(* Logix 5000 project; controller Hose_HP_Test_Rig_V1 vendor 1 type 14 code 149 rev 32.11; software revision 32.00; part 2 of 10 *)

ADD_ON_INSTRUCTION SA_SOL_FWD_RET_SEQ   (* revision 1.0 *)
VAR_INPUT
   SA_SOL_SEQ : DINT; {required}
END_VAR
VAR_OUTPUT
   SA_SOL_SOL : BOOL; {required}
END_VAR
VAR_INPUT
   SA_SOL_PS : BOOL; {required}
END_VAR
VAR_OUTPUT
   SA_FWD_PS_OK : BOOL; {access None, required}
   SA_SOL_PS_FLT : BOOL; {required}
END_VAR
VAR_INPUT
   FLT_RST_PB : BOOL; {required}
   MSG_CODE : DINT; {required}
   FLT_CODE : DINT; {required}
END_VAR
VAR_OUTPUT
   ERROR_CODE : DINT; {required}
END_VAR
VAR_INPUT
   SEQ_NO : DINT;
   SA_RET_PS : BOOL; {required}
END_VAR
VAR_OUTPUT
   SA_RET_PS_OK : BOOL; {required}
END_VAR
VAR
   SA_SOL_SEQ_ON : BOOL; {access None}
   DA_SOL_PS_FAULT : TIMER; {access None}
   SA_SOL_PS_FAULT : TIMER := (PRE := 3000); {access None}
END_VAR

ROUTINE Logic   (* ladder *)
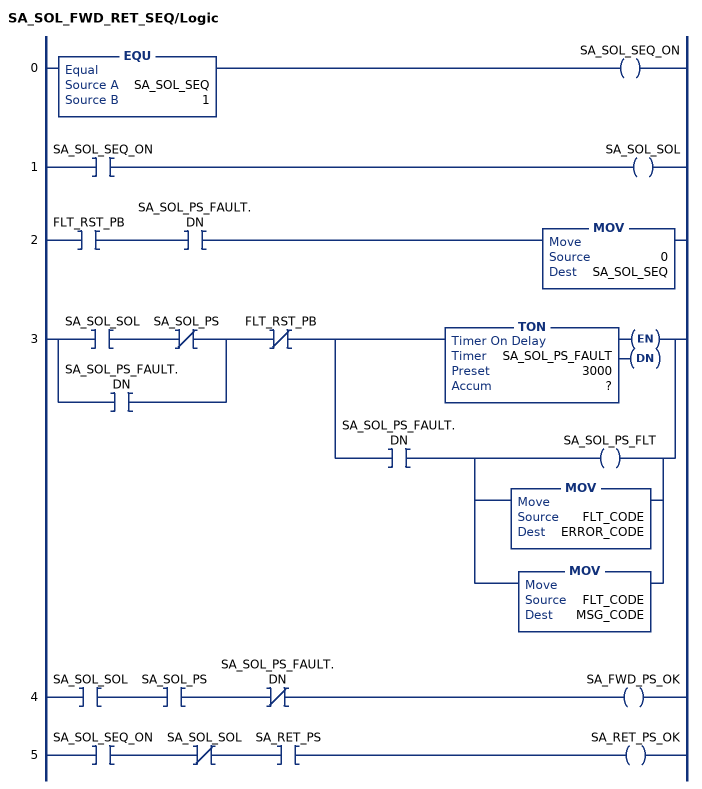
   0: EQU(SA_SOL_SEQ,1)OTE(SA_SOL_SEQ_ON);
   1: XIC(SA_SOL_SEQ_ON)OTE(SA_SOL_SOL);
   2: XIC(FLT_RST_PB)XIC(SA_SOL_PS_FAULT.DN)MOV(0,SA_SOL_SEQ);
   3: [XIC(SA_SOL_SOL) XIO(SA_SOL_PS) ,XIC(SA_SOL_PS_FAULT.DN) ]XIO(FLT_RST_PB)[TON(SA_SOL_PS_FAULT,?,?) ,XIC(SA_SOL_PS_FAULT.DN) [OTE(SA_SOL_PS_FLT) ,MOV(FLT_CODE,ERROR_CODE) ,MOV(FLT_CODE,MSG_CODE) ] ];
   4: XIC(SA_SOL_SOL)XIC(SA_SOL_PS)XIO(SA_SOL_PS_FAULT.DN)OTE(SA_FWD_PS_OK);
   5: XIC(SA_SOL_SEQ_ON)XIO(SA_SOL_SOL)XIC(SA_RET_PS)OTE(SA_RET_PS_OK);
END_ROUTINE
END_ADD_ON_INSTRUCTION

ADD_ON_INSTRUCTION SCP   (* revision 1.0 *)
VAR_OUTPUT
   Y : REAL; {access Read Only, required}
END_VAR
VAR_INPUT
   X : REAL; {required}
   X1 : REAL; {required}
   X2 : REAL; {required}
   Y1 : REAL; {required}
   Y2 : REAL; {required}
   C : REAL; {required}
END_VAR

ROUTINE Logic   (* structured text *)
   Y:=((X-X1)*((Y2-Y1)/(X2-X1))+Y1)+C;
END_ROUTINE
END_ADD_ON_INSTRUCTION

ADD_ON_INSTRUCTION SEQ_START_AND_FILL   (* revision 1.0 *)
VAR_INPUT
   SET_SEQ_NO : DINT; {required}
END_VAR
VAR_IN_OUT
   CURR_SEQ_NO : DINT; {required}
END_VAR
VAR_OUTPUT
   EXHS_VAL_ON : BOOL; {required}
   TEST_VAL_ON : BOOL; {required}
END_VAR
VAR_INPUT
   TEST_VAL_OFF : BOOL; {required}
   FAULTED : BOOL; {required}
   RST_TEST_VAL_OFF : BOOL; {required}
   EXHS_VAL_OFF : BOOL; {required}
   RST_EXHS_VAL_OFF : BOOL; {required}
END_VAR
VAR_IN_OUT
   TEST_STS : DINT; {required}
END_VAR
VAR_INPUT
   NEXT_SEQ_NO : DINT; {required}
END_VAR
VAR
   SEQ_START : BOOL; {access None}
   ONS1 : BOOL; {access None}
   ONS2 : BOOL; {access None}
   TEST_VAL_ON_DEL : TIMER := (PRE := 500); {access None}
   ONS3 : BOOL; {access None}
   EXHS_VAL_DEL : TIMER := (PRE := 250); {access None}
END_VAR

ROUTINE Logic   (* ladder *)
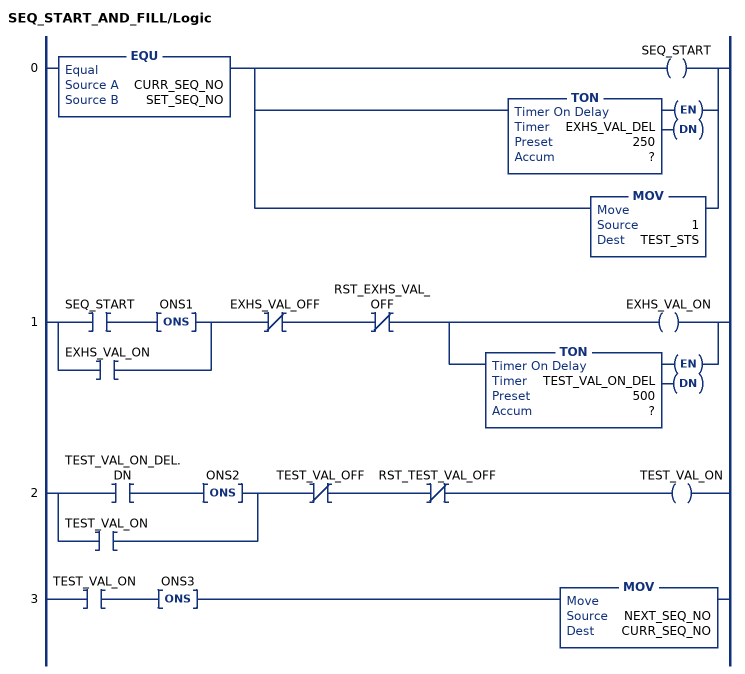
   0: EQU(CURR_SEQ_NO,SET_SEQ_NO)[OTE(SEQ_START) ,TON(EXHS_VAL_DEL,?,?) ,MOV(1,TEST_STS) ];
   1: [XIC(SEQ_START) ONS(ONS1) ,XIC(EXHS_VAL_ON) ]XIO(EXHS_VAL_OFF)XIO(RST_EXHS_VAL_OFF)[OTE(EXHS_VAL_ON) ,TON(TEST_VAL_ON_DEL,?,?) ];
   2: [XIC(TEST_VAL_ON_DEL.DN) ONS(ONS2) ,XIC(TEST_VAL_ON) ]XIO(TEST_VAL_OFF)XIO(RST_TEST_VAL_OFF)OTE(TEST_VAL_ON);
   3: XIC(TEST_VAL_ON)ONS(ONS3)MOV(NEXT_SEQ_NO,CURR_SEQ_NO);
END_ROUTINE
END_ADD_ON_INSTRUCTION

ADD_ON_INSTRUCTION SETTING_MODE   (* revision 1.0 *)
VAR_IN_OUT
   CURRENT_SCREEN : DINT; {required}
END_VAR
VAR_INPUT
   SET_MODE_SCREEN : DINT; {required}
   CALB_MODE_SCREEN : BOOL; {required}
END_VAR
VAR_OUTPUT
   SET_MODE_SEL : BOOL; {required}
END_VAR
VAR_INPUT
   LH_START_PB : BOOL; {required}
   TOP_CLAMP_SEL : BOOL; {required}
END_VAR
VAR_OUTPUT
   TOP_CLAMP_SET : BOOL; {required}
   TOP_DECLAMP_SET : BOOL; {required}
END_VAR
VAR_INPUT
   RST_SEQ_ON : BOOL; {required}
   BOTTOM_CLAMP_SEL : BOOL; {required}
END_VAR
VAR_OUTPUT
   BOTTOM_DECLAMP_SET : BOOL; {required}
   BOTTOM_CLAMP_SET : BOOL; {required}
END_VAR
VAR_INPUT
   DOOR_CLOSE_SEL : BOOL; {required}
END_VAR
VAR_OUTPUT
   DOOR_CLOSE_SET : BOOL; {required}
   DOOR_OPEN_SET : BOOL; {required}
END_VAR
VAR
   ONS1 : BOOL; {access None}
   SET_PB_ONS : BOOL; {access None}
   TOP_DECLAMP_OFF_DEL : TIMER := (PRE := 250); {access None}
   BOTTOM_DECLAMP_OFF_DEL : TIMER := (PRE := 250); {access None}
   DOOR_OPEN_OFF_DEL : TIMER := (PRE := 250); {access None}
   ons2 : BOOL; {access None}
END_VAR

ROUTINE Logic   (* ladder *)
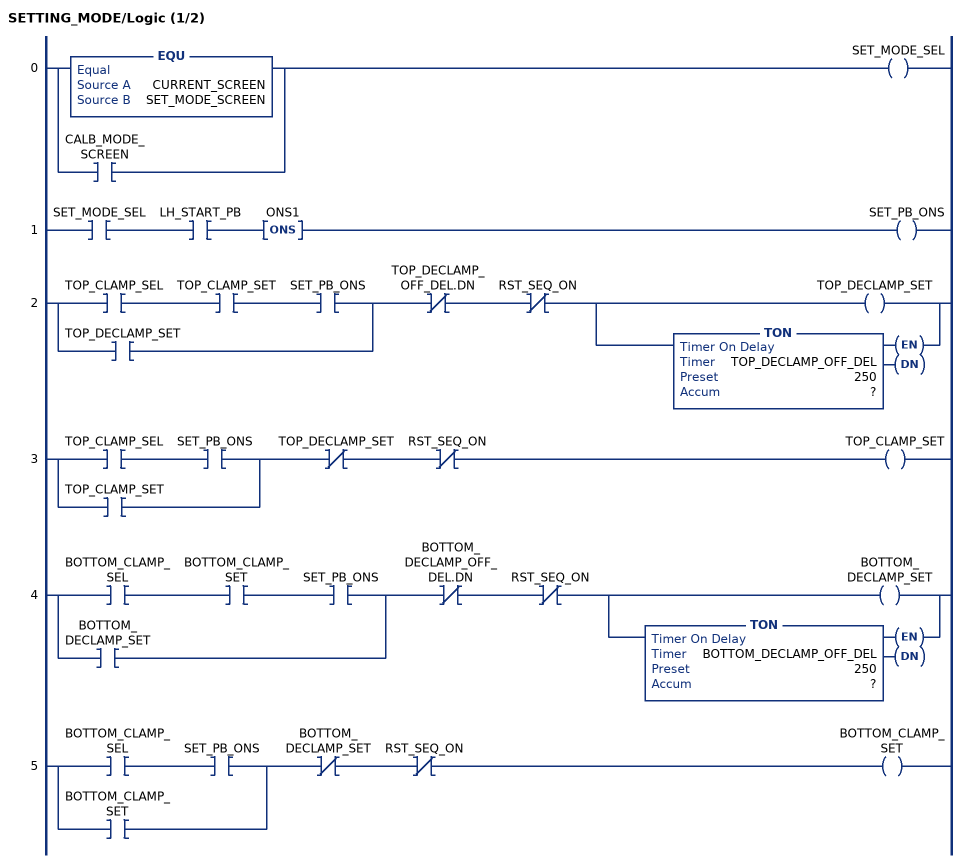
   0: [EQU(CURRENT_SCREEN,SET_MODE_SCREEN) ,XIC(CALB_MODE_SCREEN) ]OTE(SET_MODE_SEL);
   1: XIC(SET_MODE_SEL)XIC(LH_START_PB)ONS(ONS1)OTE(SET_PB_ONS);
   2: [XIC(TOP_CLAMP_SEL) XIC(TOP_CLAMP_SET) XIC(SET_PB_ONS) ,XIC(TOP_DECLAMP_SET) ]XIO(TOP_DECLAMP_OFF_DEL.DN)XIO(RST_SEQ_ON)[OTE(TOP_DECLAMP_SET) ,TON(TOP_DECLAMP_OFF_DEL,?,?) ];
   3: [XIC(TOP_CLAMP_SEL) XIC(SET_PB_ONS) ,XIC(TOP_CLAMP_SET) ]XIO(TOP_DECLAMP_SET)XIO(RST_SEQ_ON)OTE(TOP_CLAMP_SET);
   4: [XIC(BOTTOM_CLAMP_SEL) XIC(BOTTOM_CLAMP_SET) XIC(SET_PB_ONS) ,XIC(BOTTOM_DECLAMP_SET) ]XIO(BOTTOM_DECLAMP_OFF_DEL.DN)XIO(RST_SEQ_ON)[OTE(BOTTOM_DECLAMP_SET) ,TON(BOTTOM_DECLAMP_OFF_DEL,?,?) ];
   5: [XIC(BOTTOM_CLAMP_SEL) XIC(SET_PB_ONS) ,XIC(BOTTOM_CLAMP_SET) ]XIO(BOTTOM_DECLAMP_SET)XIO(RST_SEQ_ON)OTE(BOTTOM_CLAMP_SET);
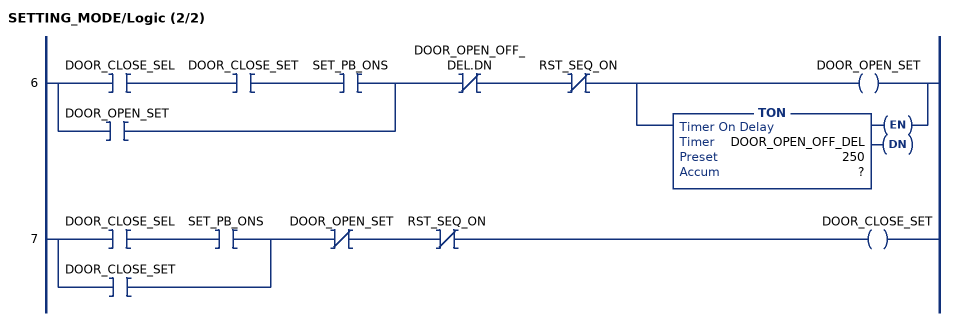
   6: [XIC(DOOR_CLOSE_SEL) XIC(DOOR_CLOSE_SET) XIC(SET_PB_ONS) ,XIC(DOOR_OPEN_SET) ]XIO(DOOR_OPEN_OFF_DEL.DN)XIO(RST_SEQ_ON)[OTE(DOOR_OPEN_SET) ,TON(DOOR_OPEN_OFF_DEL,?,?) ];
   7: [XIC(DOOR_CLOSE_SEL) XIC(SET_PB_ONS) ,XIC(DOOR_CLOSE_SET) ]XIO(DOOR_OPEN_SET)XIO(RST_SEQ_ON)OTE(DOOR_CLOSE_SET);
END_ROUTINE
END_ADD_ON_INSTRUCTION

ADD_ON_INSTRUCTION STAMP_SEQ   (* revision 1.0 *)
VAR_INPUT
   SET_SEQ_NO : DINT; {required}
END_VAR
VAR_IN_OUT
   CUR_SEQ_NO : DINT; {required}
END_VAR
VAR_OUTPUT
   STAMP_FWD_SOL : BOOL; {required}
END_VAR
VAR_INPUT
   STAMP_FWD_PS : BOOL; {required}
END_VAR
VAR_OUTPUT
   STAMP_FWD_OK : BOOL; {required}
   STAMP_NOT_FWD : BOOL; {required}
   STAMP_RET_OK : BOOL;
END_VAR
VAR_INPUT
   FLT_RST_PB : BOOL; {required}
   FAULTED : BOOL; {required}
   FLT_CODE : DINT; {required}
END_VAR
VAR_IN_OUT
   ERROR_CODE : DINT; {required}
END_VAR
VAR_INPUT
   RUN_CODE : DINT; {required}
END_VAR
VAR_IN_OUT
   MSG : DINT; {required}
END_VAR
VAR_INPUT
   NEXT_SEQ_NO : DINT; {required}
END_VAR
VAR
   STAMP_SEQ : BOOL; {access None}
   STAMP_PS_CHK_DEL : TIMER := (PRE := 3000); {access None}
   STAMP_PS_FWD_CHK : TIMER := (PRE := 500); {access None}
END_VAR

ROUTINE Logic   (* ladder *)
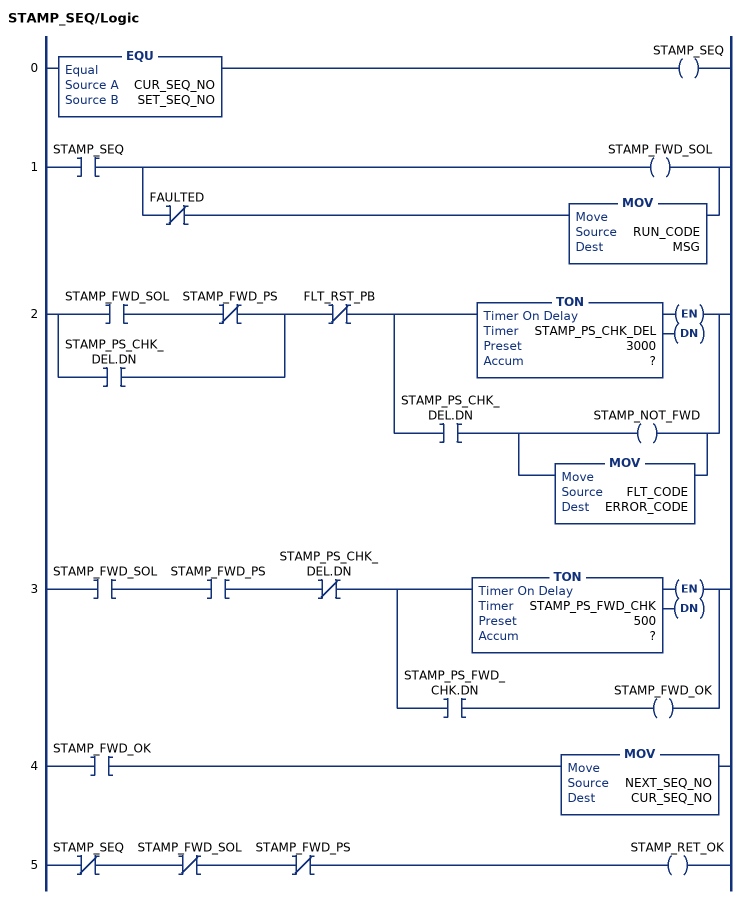
   0: EQU(CUR_SEQ_NO,SET_SEQ_NO)OTE(STAMP_SEQ);
   1: XIC(STAMP_SEQ)[OTE(STAMP_FWD_SOL) ,XIO(FAULTED) MOV(RUN_CODE,MSG) ];
   2: [XIC(STAMP_FWD_SOL) XIO(STAMP_FWD_PS) ,XIC(STAMP_PS_CHK_DEL.DN) ]XIO(FLT_RST_PB)[TON(STAMP_PS_CHK_DEL,?,?) ,XIC(STAMP_PS_CHK_DEL.DN) [OTE(STAMP_NOT_FWD) ,MOV(FLT_CODE,ERROR_CODE) ] ];
   3: XIC(STAMP_FWD_SOL)XIC(STAMP_FWD_PS)XIO(STAMP_PS_CHK_DEL.DN)[TON(STAMP_PS_FWD_CHK,?,?) ,XIC(STAMP_PS_FWD_CHK.DN) OTE(STAMP_FWD_OK) ];
   4: XIC(STAMP_FWD_OK)MOV(NEXT_SEQ_NO,CUR_SEQ_NO);
   5: XIO(STAMP_SEQ)XIO(STAMP_FWD_SOL)XIO(STAMP_FWD_PS)OTE(STAMP_RET_OK);
END_ROUTINE
END_ADD_ON_INSTRUCTION

ADD_ON_INSTRUCTION TEST_TAIL_END   (* revision 1.0 *)
VAR_INPUT
   SET_SEQ_NO : DINT; {required}
END_VAR
VAR_IN_OUT
   CUR_SEQ_NO : DINT; {required}
END_VAR
VAR_INPUT
   STN_ON : BOOL; {required}
   AUTO_MODE : BOOL; {required}
   POKAYOKE_NOT_DONE : BOOL; {required}
   PYOKE_LT : BOOL; {required}
   STAB_HIGH : BOOL; {required}
   STAB_LOW : BOOL; {required}
END_VAR
VAR_OUTPUT
   LT_COMPLETED : BOOL; {required}
END_VAR
VAR_INPUT
   LT_DROP_OK : BOOL; {required}
   DROP_NOK : BOOL; {required}
END_VAR
VAR_IN_OUT
   LT_POKEYOKE : DINT; {required}
   TEST_STS : DINT; {required}
END_VAR
VAR_INPUT
   NEXT_SEQ_NO : DINT; {required}
END_VAR

ROUTINE Logic   (* ladder *)
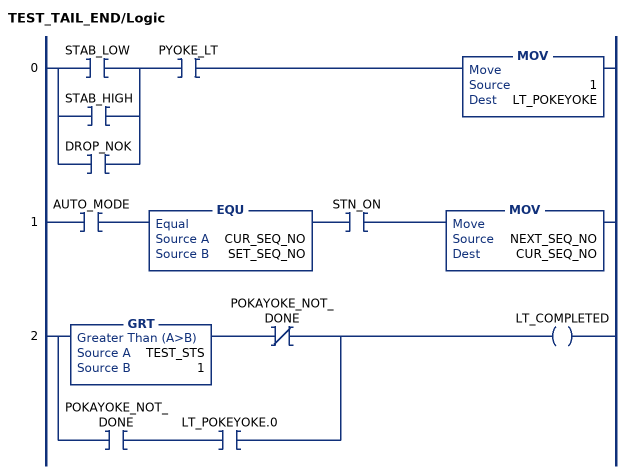
   0: [XIC(STAB_LOW) ,XIC(STAB_HIGH) ,XIC(DROP_NOK) ]XIC(PYOKE_LT)MOV(1,LT_POKEYOKE);
   1: XIC(AUTO_MODE)EQU(CUR_SEQ_NO,SET_SEQ_NO)XIC(STN_ON)MOV(NEXT_SEQ_NO,CUR_SEQ_NO);
   2: [GRT(TEST_STS,1) XIO(POKAYOKE_NOT_DONE) ,XIC(POKAYOKE_NOT_DONE) XIC(LT_POKEYOKE.0) ]OTE(LT_COMPLETED);
END_ROUTINE
END_ADD_ON_INSTRUCTION

ADD_ON_INSTRUCTION TOP_DECLAMP   (* revision 1.0 *)
VAR_INPUT
   SET_SEQ_NO : DINT; {required}
END_VAR
VAR_IN_OUT
   CUR_SEQ_NO : DINT; {required}
END_VAR
VAR_INPUT
   TEST_ON : BOOL; {required}
   FAULTED : BOOL; {required}
END_VAR
VAR_OUTPUT
   TOP_DECLAMP_AUTO : BOOL; {required}
   TOP_DECLAMP_OK : BOOL; {required}
END_VAR
VAR_INPUT
   TOP_CLAMP_PS : BOOL; {required}
   TOP_NOT_DECLAMPED : BOOL; {required}
   CONSTRICTION : BOOL; {required}
   NEXT_SEQ_NO : DINT; {required}
   END_SEQ_NO : DINT; {required}
END_VAR
VAR
   TOP_DECLAMP_SEQ_AUTO : BOOL; {access None}
   ONS1 : BOOL; {access None}
   TOP_DECLAMP_CHK_DEL : TIMER := (PRE := 500); {access None}
END_VAR

ROUTINE Logic   (* ladder *)
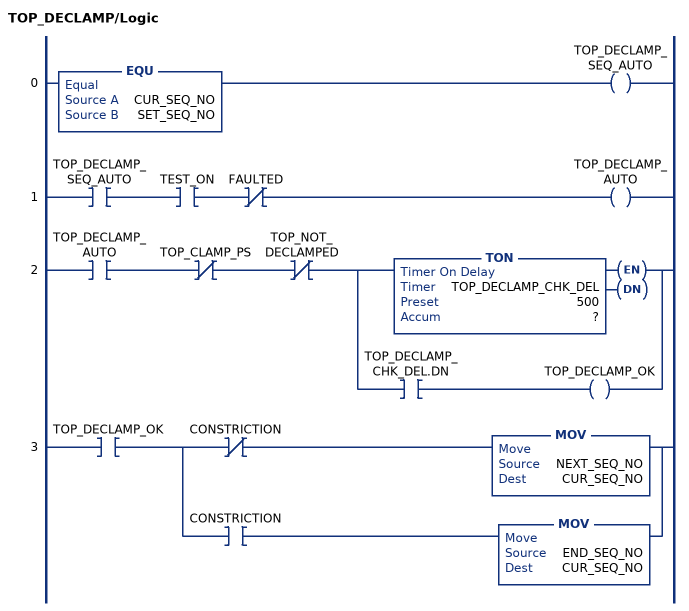
   0: EQU(CUR_SEQ_NO,SET_SEQ_NO)OTE(TOP_DECLAMP_SEQ_AUTO);
   1: XIC(TOP_DECLAMP_SEQ_AUTO)XIC(TEST_ON)XIO(FAULTED)OTE(TOP_DECLAMP_AUTO);
   2: XIC(TOP_DECLAMP_AUTO)XIO(TOP_CLAMP_PS)XIO(TOP_NOT_DECLAMPED)[TON(TOP_DECLAMP_CHK_DEL,?,?) ,XIC(TOP_DECLAMP_CHK_DEL.DN) OTE(TOP_DECLAMP_OK) ];
   3: XIC(TOP_DECLAMP_OK)[XIO(CONSTRICTION) MOV(NEXT_SEQ_NO,CUR_SEQ_NO) ,XIC(CONSTRICTION) MOV(END_SEQ_NO,CUR_SEQ_NO) ];
END_ROUTINE
END_ADD_ON_INSTRUCTION

ADD_ON_INSTRUCTION TS_TIMEOUT   (* revision 1.0 *)
VAR_IN_OUT
   TS_STS : DINT; {required}
END_VAR
VAR_INPUT
   CHECK_TRACE_STS : BOOL; {required}
   RETEST : BOOL; {required}
END_VAR
VAR_IN_OUT
   MSG : DINT; {required}
END_VAR
VAR_OUTPUT
   TS_TIMEOUT_FLT : BOOL; {access Read Only, required}
END_VAR
VAR
   TS_TIMEOUT : TIMER := (PRE := 3000); {access None}
END_VAR

ROUTINE Logic   (* ladder *)
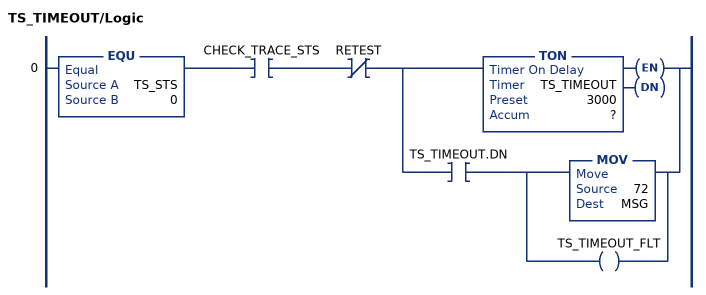
   0: EQU(TS_STS,0)XIC(CHECK_TRACE_STS)XIO(RETEST)[TON(TS_TIMEOUT,?,?) ,XIC(TS_TIMEOUT.DN) [MOV(72,MSG) ,OTE(TS_TIMEOUT_FLT) ] ];
END_ROUTINE
END_ADD_ON_INSTRUCTION

VAR_GLOBAL   (* controller tags *)
   ABORT_STN1 : BOOL;
   ABORT_STN2 : BOOL;
   ABORT_STN3 : BOOL;
   ABORT_STN4 : BOOL;
   ACT_DROP_STN1 : REAL := 0.49569702;
   ACT_DROP_STN2 : REAL := 0.5277252;
   ACT_DROP_STN3 : REAL := 0.5121765;
   ACT_DROP_STN4 : REAL := 0.4958496;
   ACT_PR_STN1 : REAL := -0.05;
   ACT_PR_STN2 : REAL := -0.015992021;
   ACT_PR_STN3 : REAL;
   ACT_PR_STN4 : REAL := 0.015994694;
   ACT_TRAVEL : REAL := 9187.228;
   AUTO_DOOR_OPEN_BLK_STN1 : DA_SOL_RET_SEQ := (FWD_SOL_PS := 1, RUN_CODE := 3, FLT_CODE := 18, SET_SEQ_NO := 97);
   AUTO_DOOR_OPEN_BLK_STN2 : DA_SOL_RET_SEQ := (FWD_SOL_PS := 1, RUN_CODE := 3, FLT_CODE := 18, SET_SEQ_NO := 97);
   AUTO_DOOR_OPEN_BLK_STN3 : DA_SOL_RET_SEQ := (FWD_SOL_PS := 1, RUN_CODE := 3, FLT_CODE := 18, SET_SEQ_NO := 97);
   AUTO_DOOR_OPEN_BLK_STN4 : DA_SOL_RET_SEQ := (FWD_SOL_PS := 1, RUN_CODE := 3, FLT_CODE := 18, SET_SEQ_NO := 97);
   AUTO_DOOR_OPEN_ON : BOOL;
   AUTO_DOOR_OPEN_ON_STN2 : BOOL;
   AUTO_DOOR_OPEN_ON_STN3 : BOOL;
   AUTO_DOOR_OPEN_ON_STN4 : BOOL;
   AUTO_DOOR_OPEN_SEQ : DINT;
   AUTO_DOOR_OPEN_SEQ_STN2 : DINT;
   AUTO_DOOR_OPEN_SEQ_STN3 : DINT;
   AUTO_DOOR_OPEN_SEQ_STN4 : DINT;
   AUTO_MODE_STN1 : BOOL;
   AUTO_MODE_STN2 : BOOL;
   AUTO_MODE_STN3 : BOOL;
   AUTO_MODE_STN4 : BOOL;
   AUTO_TEST_ON_STN1 : BOOL;
   AUTO_TEST_ON_STN2 : BOOL;
   AUTO_TEST_ON_STN3 : BOOL;
   AUTO_TEST_ON_STN4 : BOOL;
   AUTO_TEST_ON_STN5 : BOOL;
   AUTO_TEST_OVER_DEL : TIMER := (PRE := 500);
   AUTO_TEST_OVER_STN1 : BOOL;
   AUTO_TEST_OVER_STN2 : BOOL;
   AUTO_TEST_OVER_STN3 : BOOL;
   AUTO_TEST_OVER_STN4 : BOOL;
   AUTO_TEST_SEL_STN1 : BOOL := 1;
   AUTO_TEST_SEL_STN2 : BOOL := 1;
   AUTO_TEST_SEL_STN3 : BOOL := 1;
   AUTO_TEST_SEL_STN4 : BOOL := 1;
   BIN_MSG : DINT;
   BOTTOM_CLAMP_2BPR_HIGH : BOOL;
   BOTTOM_CLAMP_2BPR_HIGH_STN2 : BOOL;
   BOTTOM_CLAMP_2BPR_HIGH_STN3 : BOOL;
   BOTTOM_CLAMP_2BPR_HIGH_STN4 : BOOL;
   BOTTOM_CLAMP_2BPR_LOW : BOOL;
   BOTTOM_CLAMP_2BPR_LOW_STN2 : BOOL;
   BOTTOM_CLAMP_2BPR_LOW_STN3 : BOOL;
   BOTTOM_CLAMP_2BPR_LOW_STN4 : BOOL;
   BOTTOM_CLAMP_4BPR_HIGH : BOOL;
   BOTTOM_CLAMP_4BPR_HIGH_STN2 : BOOL;
   BOTTOM_CLAMP_4BPR_HIGH_STN3 : BOOL;
   BOTTOM_CLAMP_4BPR_HIGH_STN4 : BOOL;
   BOTTOM_CLAMP_4BPR_LOW : BOOL;
   BOTTOM_CLAMP_4BPR_LOW_STN2 : BOOL;
   BOTTOM_CLAMP_4BPR_LOW_STN3 : BOOL;
   BOTTOM_CLAMP_4BPR_LOW_STN4 : BOOL;
   BOTTOM_CLAMP_AUTO_STN1 : BOOL;
   BOTTOM_CLAMP_AUTO_STN2 : BOOL;
   BOTTOM_CLAMP_AUTO_STN3 : BOOL;
   BOTTOM_CLAMP_AUTO_STN4 : BOOL;
   BOTTOM_CLAMP_BLK_STN1 : DA_SOL_FWD_SEQ := (RUN_CODE := 7, FLT_CODE := 9, NEXT_SEQ_NO := 19);
   BOTTOM_CLAMP_BLK_STN2 : DA_SOL_FWD_SEQ := (RUN_CODE := 7, FLT_CODE := 9, NEXT_SEQ_NO := 20);
   BOTTOM_CLAMP_BLK_STN3 : DA_SOL_FWD_SEQ := (RUN_CODE := 7, FLT_CODE := 9, NEXT_SEQ_NO := 20);
   BOTTOM_CLAMP_BLK_STN4 : DA_SOL_FWD_SEQ := (RUN_CODE := 7, FLT_CODE := 9, NEXT_SEQ_NO := 20);
   BOTTOM_CLAMP_C : REAL;
   BOTTOM_CLAMP_FAULT_STN1 : BOOL;
   BOTTOM_CLAMP_FAULT_STN2 : BOOL;
   BOTTOM_CLAMP_FAULT_STN3 : BOOL;
   BOTTOM_CLAMP_FAULT_STN4 : BOOL;
   BOTTOM_CLAMP_OK_STN1 : BOOL;
   BOTTOM_CLAMP_OK_STN2 : BOOL;
   BOTTOM_CLAMP_OK_STN3 : BOOL;
   BOTTOM_CLAMP_OK_STN4 : BOOL;
   BOTTOM_CLAMP_PR : REAL := 4.2651687;
   BOTTOM_CLAMP_PR_CHK : TIMER := (PRE := 1000);
   BOTTOM_CLAMP_PR_DEL : TIMER := (PRE := 6000);
   BOTTOM_CLAMP_PR_SEL : BOOL := 1;
   BOTTOM_CLAMP_PR_SEL_SET : BOOL;
   BOTTOM_CLAMP_PR_SEL_SOL : ALIAS FOR REM:O.Data[1].7;
   BOTTOM_CLAMP_PR_SEQ : CLAMP_FAULT := (CLAMP_PR_SEL := 1, CLAMP_PR := 4, CLAMP_2BAR_LL := 0.1, CLAMP_2BAR_HL := 3.5, CLAMP_4BAR_LL := 0.1, CLAMP_4BAR_HL := 4.5);
   BOTTOM_CLAMP_PS_STN1 : ALIAS FOR Local:1:I.Data.13;
   BOTTOM_CLAMP_PS_STN2 : ALIAS FOR Local:2:I.Data.2;
   BOTTOM_CLAMP_PS_STN3 : ALIAS FOR Local:2:I.Data.7;
   BOTTOM_CLAMP_PS_STN4 : ALIAS FOR Local:2:I.Data.12;
   BOTTOM_CLAMP_SEL_STN1 : BOOL;
   BOTTOM_CLAMP_SEL_STN2 : BOOL;
   BOTTOM_CLAMP_SEL_STN3 : BOOL;
   BOTTOM_CLAMP_SEL_STN4 : BOOL;
   BOTTOM_CLAMP_SEQ_STN1 : DINT;
   BOTTOM_CLAMP_SEQ_STN2 : DINT;
   BOTTOM_CLAMP_SEQ_STN3 : DINT;
   BOTTOM_CLAMP_SEQ_STN4 : DINT;
   BOTTOM_CLAMP_SET_STN1 : BOOL;
   BOTTOM_CLAMP_SET_STN2 : BOOL;
   BOTTOM_CLAMP_SET_STN3 : BOOL;
   BOTTOM_CLAMP_SET_STN4 : BOOL;
   BOTTOM_CLAMP_SOL_STN1 : ALIAS FOR Local:1:O.Data.4;
   BOTTOM_CLAMP_SOL_STN2 : ALIAS FOR Local:1:O.Data.12;
   BOTTOM_CLAMP_SOL_STN3 : ALIAS FOR Local:3:O.Data.4;
   BOTTOM_CLAMP_SOL_STN4 : ALIAS FOR Local:3:O.Data.12;
   BOTTOM_CLAMP_X : REAL := 4.263;
   BOTTOM_CLAMP_X1 : REAL;
   BOTTOM_CLAMP_X2 : REAL := 5.898;
   BOTTOM_CLAMP_Y1 : REAL;
   BOTTOM_CLAMP_Y2 : REAL := 5.901;
   BOTTOM_DECLAMP_AUTO_STN1 : BOOL;
   BOTTOM_DECLAMP_AUTO_STN2 : BOOL;
   BOTTOM_DECLAMP_AUTO_STN3 : BOOL;
   BOTTOM_DECLAMP_AUTO_STN4 : BOOL;
   BOTTOM_DECLAMP_OK_STN1 : BOOL;
   BOTTOM_DECLAMP_OK_STN2 : BOOL;
   BOTTOM_DECLAMP_OK_STN3 : BOOL;
   BOTTOM_DECLAMP_OK_STN4 : BOOL;
   BOTTOM_DECLAMP_SEQ_STN1 : DINT;
   BOTTOM_DECLAMP_SEQ_STN2 : DINT;
   BOTTOM_DECLAMP_SEQ_STN3 : DINT;
   BOTTOM_DECLAMP_SEQ_STN4 : DINT;
   BOTTOM_DECLAMP_SET_STN1 : BOOL;
   BOTTOM_DECLAMP_SET_STN2 : BOOL;
   BOTTOM_DECLAMP_SET_STN3 : BOOL;
   BOTTOM_DECLAMP_SET_STN4 : BOOL;
   BOTTOM_DECLAMP_SOL_STN1 : ALIAS FOR REM:O.Data[0].3;
   BOTTOM_DECLAMP_SOL_STN2 : ALIAS FOR REM:O.Data[0].5;
   BOTTOM_DECLAMP_SOL_STN3 : ALIAS FOR REM:O.Data[0].7;
   BOTTOM_DECLAMP_SOL_STN4 : ALIAS FOR REM:O.Data[1].1;
   BOTTOM_DECLMP_BLK_STN1 : DA_SOL_RET_SEQ := (RUN_CODE := 8, FLT_CODE := 41, SET_SEQ_NO := 57);
   BOTTOM_DECLMP_BLK_STN2 : DA_SOL_RET_SEQ := (RUN_CODE := 8, FLT_CODE := 41, SET_SEQ_NO := 57);
   BOTTOM_DECLMP_BLK_STN3 : DA_SOL_RET_SEQ := (RUN_CODE := 8, FLT_CODE := 41, SET_SEQ_NO := 57);
   BOTTOM_DECLMP_BLK_STN4 : DA_SOL_RET_SEQ := (RUN_CODE := 8, FLT_CODE := 41, SET_SEQ_NO := 57);
   BOTTOM_DECLMP_CBLK_STN1 : BOTTOM_DECLAMP;
   BOTTOM_NOT_CLAMPED_STN1 : BOOL;
   BOTTOM_NOT_CLAMPED_STN2 : BOOL;
   BOTTOM_NOT_CLAMPED_STN4 : BOOL;
   BOTTOM_NOT_DECLAMPED_STN1 : BOOL;
   BOTTOM_NOT_DECLAMPED_STN2 : BOOL;
   BOTTOM_NOT_DECLAMPED_STN3 : BOOL;
   BOTTOM_NOT_DECLAMPED_STN4 : BOOL;
   BOTTOM_PR_SCL : SCP := (Y := 4.2651687, X := 4.263, X2 := 5.898, Y2 := 5.901);
   BUZZER_STN1 : ALIAS FOR Local:3:O.Data.20;
   BUZZER_STN2 : ALIAS FOR Local:3:O.Data.24;
   BUZZER_STN3 : ALIAS FOR Local:3:O.Data.29;
   BUZZER_STN4 : ALIAS FOR REM:O.Data[0].1;
   CALB_START_PB_ONS_STN1 : BOOL;
   CALB_START_PB_ONS_STN2 : BOOL;
   CALB_START_PB_ONS_STN3 : BOOL;
   CALB_START_PB_ONS_STN4 : BOOL;
   CHECK_TRACE_STS_STN1 : BOOL;
   CHECK_TRACE_STS_STN2 : BOOL;
   CHECK_TRACE_STS_STN3 : BOOL;
   CHECK_TRACE_STS_STN4 : BOOL;
   CLAMP_2BAR_HL : REAL := 3.5;
   CLAMP_2BAR_LL : REAL := 0.1;
   CLAMP_4BAR_HL : REAL := 4.5;
   CLAMP_4BAR_LL : REAL := 0.1;
   CLR_FAIL_ONS_STN1 : BOOL;
   CLR_FAIL_ONS_STN2 : BOOL;
   CLR_FAIL_ONS_STN3 : BOOL;
   CLR_FAIL_ONS_STN4 : BOOL;
   CLR_FLT_ONS_STN1 : BOOL;
   CLR_ONS_STN1 : BOOL;
   CLR_ONS_STN2 : BOOL;
   CLR_ONS_STN3 : BOOL;
   CLR_ONS_STN4 : BOOL;
   COMP_FAULT_STN1 : BOOL;
   COMP_FAULT_STN2 : BOOL;
   COMP_FAULT_STN3 : BOOL;
   COMP_FAULT_STN4 : BOOL;
   CONS_CALB_OFF_STN1 : BOOL;
   CONS_CALB_OFF_STN2 : BOOL;
   CONS_CALB_OFF_STN3 : BOOL;
   CONS_CALB_OFF_STN4 : BOOL;
   CONS_CALB_ON_STN1 : BOOL;
   CONS_CALB_ON_STN2 : BOOL;
   CONS_CALB_ON_STN3 : BOOL;
   CONS_CALB_ON_STN4 : BOOL;
   CONS_CALB_TARRED_STN1 : BOOL;
   CONS_CALB_TARRED_STN2 : BOOL;
   CONS_CALB_TARRED_STN3 : BOOL;
   CONS_CALB_TARRED_STN4 : BOOL;
   CONS_DUMMIT_VAR : REAL := 0.004;
   CONS_FAIL_COUNT_STN1 : DINT;
   CONS_FAIL_COUNT_STN2 : DINT;
   CONS_FAIL_COUNT_STN3 : DINT;
   CONS_FAIL_COUNT_STN4 : DINT;
   CONS_FAIL_COUNTER_STN1 : COUNTER := (PRE := 9999);
   CONS_FAIL_COUNTER_STN2 : COUNTER := (PRE := 9999);
   CONS_FAIL_COUNTER_STN3 : COUNTER := (PRE := 9999);
   CONS_FAIL_COUNTER_STN4 : COUNTER := (PRE := 9999);
   CONS_FAULT_COUNTER_STN1 : COUNTER;
   CONS_FILL_BLK_STN1 : CONSTRICTION_FILL_ON_SEQ := (SET_SEQ_NO := 60, TEST_STS := 1, NEXT_SEQ_NO := 65);
   CONS_FILL_BLK_STN2 : CONSTRICTION_FILL_ON_SEQ := (SET_SEQ_NO := 60, TEST_STS := 1, NEXT_SEQ_NO := 65);
   CONS_FILL_BLK_STN3 : CONSTRICTION_FILL_ON_SEQ := (SET_SEQ_NO := 60, TEST_STS := 1, NEXT_SEQ_NO := 65);
   CONS_FILL_BLK_STN4 : CONSTRICTION_FILL_ON_SEQ := (SET_SEQ_NO := 60, TEST_STS := 1, NEXT_SEQ_NO := 65);
   CONS_FILL_HIGH_STN1 : BOOL;
   CONS_FILL_HIGH_STN2 : BOOL;
   CONS_FILL_HIGH_STN3 : BOOL;
   CONS_FILL_HIGH_STN4 : BOOL;
   CONS_FILL_HL : REAL := 2400.0;
   CONS_FILL_LL : REAL := 1800.0;
   CONS_FILL_LOW_STN1 : BOOL;
   CONS_FILL_LOW_STN2 : BOOL;
   CONS_FILL_LOW_STN3 : BOOL;
   CONS_FILL_LOW_STN4 : BOOL;
   CONS_FILL_OFF_BLK_STN1 : CONSTRICTION_FILL_OFF_SEQ := (SET_SEQ_NO := 75, NEXT_SEQ_NO := 81);
   CONS_FILL_OFF_BLK_STN2 : CONSTRICTION_FILL_OFF_SEQ := (SET_SEQ_NO := 75, NEXT_SEQ_NO := 81);
   CONS_FILL_OFF_BLK_STN3 : CONSTRICTION_FILL_OFF_SEQ := (SET_SEQ_NO := 75, NEXT_SEQ_NO := 81);
   CONS_FILL_OFF_BLK_STN4 : CONSTRICTION_FILL_OFF_SEQ := (SET_SEQ_NO := 75, NEXT_SEQ_NO := 81);
   CONS_FILL_TIME_ACT_STN1 : REAL;
   CONS_FILL_TIME_ACT_STN2 : REAL;
   CONS_FILL_TIME_ACT_STN3 : REAL;
   CONS_FILL_TIME_ACT_STN4 : REAL;
   CONS_FILL_TIME_SET : REAL;
   CONS_P2_STN1 : REAL;
   CONS_P2_STN2 : REAL;
   CONS_P2_STN3 : REAL;
   CONS_P2_STN4 : REAL;
   CONS_PR : REAL;
   CONS_PR_BLK_STN1 : PR_CHECK := (SET_SEQ := 65, ACT_PR := 2677.0298, PR_LL := 1800.0, PR_HL := 2400.0, SET_TIME := 3.0, ACT_TIME := 3.001, PR_AT_END := 2070.028, SEQ_STS_CODE := 4, RUN_CODE := 15, LIM_LOW_CODE := 18, LIM_HIGH_CODE := 19, NEXT_SEQ_NO := 66);
   CONS_PR_BLK_STN2 : PR_CHECK := (SET_SEQ := 65, ACT_PR := 2677.0298, PR_LL := 1800.0, PR_HL := 2400.0, SET_TIME := 3.0, ACT_TIME := 3.004, PR_AT_END := 2062.1184, SEQ_STS_CODE := 4, RUN_CODE := 15, LIM_LOW_CODE := 18, LIM_HIGH_CODE := 19, NEXT_SEQ_NO := 66);
   CONS_PR_BLK_STN3 : PR_CHECK := (SET_SEQ := 65, ACT_PR := 2677.0298, PR_LL := 1800.0, PR_HL := 2400.0, SET_TIME := 3.0, ACT_TIME := 3.001, PR_AT_END := 2023.3356, SEQ_STS_CODE := 4, RUN_CODE := 15, LIM_LOW_CODE := 18, LIM_HIGH_CODE := 19, NEXT_SEQ_NO := 66);
   CONS_PR_BLK_STN4 : PR_CHECK := (SET_SEQ := 65, ACT_PR := 2677.0298, PR_LL := 1800.0, PR_HL := 2400.0, SET_TIME := 3.0, ACT_TIME := 3.0, PR_AT_END := 2092.481, SEQ_STS_CODE := 4, RUN_CODE := 15, LIM_LOW_CODE := 18, LIM_HIGH_CODE := 19, NEXT_SEQ_NO := 66);
   CONS_PR_P1_STN1 : REAL := 2070.028;
   CONS_PR_P1_STN2 : REAL := 2062.1184;
   CONS_PR_P1_STN3 : REAL := 2023.3356;
   CONS_PR_P1_STN4 : REAL := 2092.481;
   CONS_PR_P2_STN2 : REAL;
   CONS_PR_P3_STN3 : REAL;
   CONS_RESULT : DINT := 2;
   CONS_RESULT_STN1 : DINT := 2;
   CONS_RESULT_STN2 : DINT := 2;
   CONS_RESULT_STN3 : DINT := 2;
   CONS_RESULT_STN4 : DINT := 2;
   CONS_STS_STN1 : DINT := 2;
   CONS_STS_STN2 : DINT := 2;
   CONS_STS_STN3 : DINT := 2;
   CONS_STS_STN4 : DINT := 2;
   CONS_TARRED_OK_STN4 : TIMER := (PRE := 10000, ACC := 10001);
   CONS_TEST_ON : BOOL := 1;
   CONS_TEST_TIME_ACT : REAL := 3.001;
   CONS_TEST_TIME_ACT_STN2 : REAL := 3.004;
   CONS_TEST_TIME_ACT_STN3 : REAL := 3.001;
   CONS_TEST_TIME_ACT_STN4 : REAL := 3.0;
   CONS_TEST_TIME_SET : REAL := 3.0;
   CONSTRICTION_BLK_STN1 : DROP_CHECK := (SET_SEQ_NO := 67, ACT_TIME := 0.005, P1 := -497.35376, PR_DIFF_LL := 50.0, PR_DIFF_HL := 500.0, ACT_DROP := 73.106445, RUN_CODE := 23, PASS_CODE := 24, FLT_CODE := 25, NEXT_SEQ_NO := 75);
   CONSTRICTION_BLK_STN2 : DROP_CHECK := (SET_SEQ_NO := 67, ACT_TIME := 0.004, P1 := -469.7915, PR_DIFF_LL := 50.0, PR_DIFF_HL := 500.0, ACT_DROP := 102.48828, RUN_CODE := 23, PASS_CODE := 24, FLT_CODE := 25, NEXT_SEQ_NO := 75);
   CONSTRICTION_BLK_STN3 : DROP_CHECK := (SET_SEQ_NO := 67, ACT_TIME := 0.004, P1 := -482.81543, PR_DIFF_LL := 50.0, PR_DIFF_HL := 500.0, ACT_DROP := 129.26184, RUN_CODE := 23, PASS_CODE := 24, FLT_CODE := 25, NEXT_SEQ_NO := 75);
   CONSTRICTION_BLK_STN4 : DROP_CHECK := (SET_SEQ_NO := 67, ACT_TIME := 0.004, P1 := -478.98828, PR_DIFF_LL := 50.0, PR_DIFF_HL := 500.0, ACT_DROP := 80.18457, RUN_CODE := 23, PASS_CODE := 24, FLT_CODE := 25, NEXT_SEQ_NO := 75);
   CONSTRICTION_CALB_SEL_STN1 : BOOL;
   CONSTRICTION_CALB_SEL_STN2 : BOOL;
   CONSTRICTION_CALB_SEL_STN3 : BOOL;
   CONSTRICTION_CALB_SEL_STN4 : BOOL;
   CONSTRICTION_FILL_OFF_STN1 : BOOL;
   CONSTRICTION_FILL_OFF_STN2 : BOOL;
   CONSTRICTION_FILL_OFF_STN3 : BOOL;
   CONSTRICTION_FILL_OFF_STN4 : BOOL;
   CONSTRICTION_FILL_VAL_STN1 : BOOL;
   CONSTRICTION_FILL_VAL_STN2 : BOOL;
   CONSTRICTION_FILL_VAL_STN3 : BOOL;
   CONSTRICTION_FILL_VAL_STN4 : BOOL;
   CONSTRICTION_NOK_STN1 : BOOL;
   CONSTRICTION_NOK_STN2 : BOOL;
   CONSTRICTION_NOK_STN3 : BOOL;
   CONSTRICTION_NOK_STN4 : BOOL;
   CONSTRICTION_OK_STN1 : BOOL;
   CONSTRICTION_OK_STN2 : BOOL;
   CONSTRICTION_OK_STN3 : BOOL;
   CONSTRICTION_OK_STN4 : BOOL;
   CONSTRICTION_SEL_STN1 : BOOL;
   CONSTRICTION_SEL_STN3 : BOOL;
   CONSTRICTION_SEL_STN4 : BOOL;
   CONSTRICTION_TEST_ON_STN1 : BOOL;
   CONSTRICTION_TEST_ON_STN2 : BOOL;
   CONSTRICTION_TEST_ON_STN3 : BOOL;
   CONSTRICTION_TEST_ON_STN4 : BOOL;
   CONSTRICTION_VALVE_SET_STN1 : BOOL;
   CONSTRICTION_VALVE_SET_STN2 : BOOL;
   CONSTRICTION_VALVE_SET_STN3 : BOOL;
   CONSTRICTION_VALVE_SET_STN4 : BOOL;
   CONSTRICTION_VALVE_STN1 : BOOL;
   CONSTRICTION_VALVE_STN2 : BOOL;
   CONSTRICTION_VALVE_STN3 : BOOL;
   CONSTRICTION_VALVE_STN4 : BOOL;
   CRIMP_PASS : ALIAS FOR Local:2:I.Data.31;
   CRIMP_PASS_TO_TRACE : DINT; {produced}
   CYCLE_START_PB_STN1 : ALIAS FOR Local:1:I.Data.2;
   CYCLE_TIME_ACT_STN1 : REAL := 41.679;
   CYCLE_TIME_ACT_STN2 : REAL := 40.582;
   CYCLE_TIME_ACT_STN3 : REAL := 40.662;
   CYCLE_TIME_ACT_STN4 : REAL := 41.107;
   CYCLE_TIMER_STN1 : TIMER := (PRE := 99999);
   CYCLE_TIMER_STN4 : TIMER := (PRE := 99999);
   DICH2_1_32 : DINT := 813761552;
   DICH_STN1 : INT := 1088;
   DICH_STN2 : INT := 1088;
   DICH_STN3 : INT := 1088;
   DICH_STN4 : INT := 1088;
   DOOR_CLAMP_SET_STN1 : SETTING_MODE := (SET_MODE_SCREEN := 17);
   DOOR_CLAMP_SET_STN2 : SETTING_MODE := (SET_MODE_SCREEN := 18);
   DOOR_CLAMP_SET_STN3 : SETTING_MODE := (SET_MODE_SCREEN := 19);
   DOOR_CLAMP_SET_STN4 : SETTING_MODE := (SET_MODE_SCREEN := 20);
   DOOR_CLOSE_ABORT_STN1 : BOOL;
   DOOR_CLOSE_ABORT_STN2 : BOOL;
   DOOR_CLOSE_ABORT_STN3 : BOOL;
   DOOR_CLOSE_ABORT_STN4 : BOOL;
   DOOR_CLOSE_AUTO_STN1 : BOOL;
   DOOR_CLOSE_AUTO_STN2 : BOOL;
   DOOR_CLOSE_AUTO_STN3 : BOOL;
   DOOR_CLOSE_AUTO_STN4 : BOOL;
   DOOR_CLOSE_BLK_STN1 : DOOR_CLOSE := (SET_SEQ_NO := 20, LH_START_PB := 1, DOOR_OPEN_RS := 1, NEXT_SEQ_NO := 24);
   DOOR_CLOSE_BLK_STN2 : DOOR_CLOSE := (SET_SEQ_NO := 20, LH_START_PB := 1, DOOR_OPEN_RS := 1, NEXT_SEQ_NO := 24);
   DOOR_CLOSE_BLK_STN3 : DOOR_CLOSE := (SET_SEQ_NO := 20, LH_START_PB := 1, DOOR_OPEN_RS := 1, NEXT_SEQ_NO := 24);
   DOOR_CLOSE_BLK_STN4 : DOOR_CLOSE := (SET_SEQ_NO := 20, LH_START_PB := 1, DOOR_OPEN_RS := 1, NEXT_SEQ_NO := 24);
   DOOR_CLOSE_OK_STN1 : BOOL;
   DOOR_CLOSE_OK_STN2 : BOOL;
   DOOR_CLOSE_OK_STN3 : BOOL;
   DOOR_CLOSE_OK_STN4 : BOOL;
   DOOR_CLOSE_RS_STN1 : ALIAS FOR Local:1:I.Data.11;
   DOOR_CLOSE_RS_STN2 : ALIAS FOR Local:2:I.Data.0;
   DOOR_CLOSE_RS_STN3 : ALIAS FOR Local:2:I.Data.5;
   DOOR_CLOSE_RS_STN4 : ALIAS FOR Local:2:I.Data.9;
   DOOR_CLOSE_SEL_STN1 : BOOL;
   DOOR_CLOSE_SEL_STN2 : BOOL;
   DOOR_CLOSE_SEL_STN3 : BOOL;
   DOOR_CLOSE_SEL_STN4 : BOOL;
   DOOR_CLOSE_SEQ_STN1 : DA_SOL_FWD_SEQ := (RUN_CODE := 2, FLT_CODE := 26, NEXT_SEQ_NO := 25);
   DOOR_CLOSE_SEQ_STN2 : DA_SOL_FWD_SEQ := (RUN_CODE := 2, FLT_CODE := 26, NEXT_SEQ_NO := 25);
   DOOR_CLOSE_SEQ_STN3 : DA_SOL_FWD_SEQ := (RUN_CODE := 2, FLT_CODE := 26, NEXT_SEQ_NO := 25);
   DOOR_CLOSE_SEQ_STN4 : DA_SOL_FWD_SEQ := (RUN_CODE := 2, FLT_CODE := 26, NEXT_SEQ_NO := 25);
   DOOR_CLOSE_SET_STN1 : BOOL;
   DOOR_CLOSE_SET_STN2 : BOOL;
   DOOR_CLOSE_SET_STN3 : BOOL;
   DOOR_CLOSE_SET_STN4 : BOOL;
   DOOR_CLOSE_SOL_STN1 : ALIAS FOR Local:1:O.Data.2;
   DOOR_CLOSE_SOL_STN2 : ALIAS FOR Local:1:O.Data.9;
   DOOR_CLOSE_SOL_STN3 : ALIAS FOR Local:3:O.Data.2;
   DOOR_CLOSE_SOL_STN4 : ALIAS FOR Local:3:O.Data.10;
   DOOR_NOT_CLOSED : BOOL;
   DOOR_NOT_CLOSED_STN2 : BOOL;
   DOOR_NOT_CLOSED_STN3 : BOOL;
   DOOR_NOT_CLOSED_STN4 : BOOL;
   DOOR_NOT_OPEN_STN1 : BOOL;
   DOOR_NOT_OPEN_STN2 : BOOL;
   DOOR_NOT_OPEN_STN3 : BOOL;
   DOOR_NOT_OPEN_STN4 : BOOL;
   DOOR_OPEN_AUTO_STN1 : BOOL;
   DOOR_OPEN_AUTO_STN2 : BOOL;
   DOOR_OPEN_AUTO_STN3 : BOOL;
   DOOR_OPEN_AUTO_STN4 : BOOL;
   DOOR_OPEN_RS_STN1 : ALIAS FOR Local:1:I.Data.10;
   DOOR_OPEN_RS_STN2 : ALIAS FOR Local:1:I.Data.15;
   DOOR_OPEN_RS_STN3 : ALIAS FOR Local:2:I.Data.4;
   DOOR_OPEN_RS_STN4 : ALIAS FOR Local:2:I.Data.10;
   DOOR_OPEN_SEQ_STN1 : DINT;
   DOOR_OPEN_SEQ_STN2 : DINT;
   DOOR_OPEN_SEQ_STN3 : DINT;
   DOOR_OPEN_SEQ_STN4 : DINT;
   DOOR_OPEN_SET_STN1 : BOOL;
   DOOR_OPEN_SET_STN2 : BOOL;
   DOOR_OPEN_SET_STN3 : BOOL;
   DOOR_OPEN_SET_STN4 : BOOL;
   DOOR_OPEN_SOL_STN1 : ALIAS FOR Local:1:O.Data.1;
   DOOR_OPEN_SOL_STN2 : ALIAS FOR Local:1:O.Data.10;
   DOOR_OPEN_SOL_STN3 : ALIAS FOR Local:3:O.Data.1;
   DOOR_OPEN_SOL_STN4 : ALIAS FOR Local:3:O.Data.9;
   DROP_CHK_SEQ_STN1 : DROP_CHECK := (SET_SEQ_NO := 45, COMPARE_TIMER_SET_TIME := 15.0, ACT_TIME := 15.001, ACT_PR := -0.05, P1 := 139.0502, PR_DIFF_HL := 1.0, ACT_DROP := 0.49569702, RUN_CODE := 14, PASS_CODE := 16, FLT_CODE := 17, NEXT_SEQ_NO := 50, P2 := 138.5545);
   DROP_CHK_SEQ_STN2 : DROP_CHECK := (SET_SEQ_NO := 45, COMPARE_TIMER_SET_TIME := 15.0, ACT_TIME := 15.001, ACT_PR := -0.015992021, P1 := 139.41847, PR_DIFF_HL := 1.0, ACT_DROP := 0.5277252, RUN_CODE := 14, PASS_CODE := 16, FLT_CODE := 17, NEXT_SEQ_NO := 50, P2 := 138.89075);
   DROP_CHK_SEQ_STN3 : DROP_CHECK := (SET_SEQ_NO := 45, COMPARE_TIMER_SET_TIME := 15.0, ACT_TIME := 15.003, P1 := 139.11847, PR_DIFF_HL := 1.0, ACT_DROP := 0.5121765, RUN_CODE := 14, PASS_CODE := 16, FLT_CODE := 17, NEXT_SEQ_NO := 50, P2 := 138.6063);
   DROP_CHK_SEQ_STN4 : DROP_CHECK := (SET_SEQ_NO := 45, COMPARE_TIMER_SET_TIME := 15.0, ACT_TIME := 15.003, ACT_PR := 0.015994694, P1 := 139.79361, PR_DIFF_HL := 1.0, ACT_DROP := 0.4958496, RUN_CODE := 14, PASS_CODE := 16, FLT_CODE := 17, NEXT_SEQ_NO := 50, P2 := 139.29776);
   DROP_NOK_STN1 : BOOL;
   DROP_NOK_STN2 : BOOL;
   DROP_NOK_STN3 : BOOL;
   DROP_NOK_STN4 : BOOL;
   DROP_OK_STN1 : BOOL;
   DROP_OK_STN2 : BOOL;
   DROP_OK_STN3 : BOOL;
   DROP_OK_STN4 : BOOL;
   DUMMIT : BOOL;
   DUPLICATE_STN1 : BOOL;
   DUPLICATE_STN2 : BOOL;
   DUPLICATE_STN3 : BOOL;
   DUPLICATE_STN4 : BOOL;
   EC_STN1 : DINT := 27;
   EC_STN2 : DINT := 17;
   EC_STN3 : DINT := 17;
   EC_STN4 : DINT := 25;
   EMG_FAULT_CLR : BOOL;
   EMG_FAULTED_STN1 : BOOL;
   EMG_FAULTED_STN2 : BOOL;
   EMG_FAULTED_STN3 : BOOL;
   EMG_FAULTED_STN4 : BOOL;
   EMG_START_PB : ALIAS FOR Local:1:I.Data.6;
   EMG_STOP_PB : ALIAS FOR Local:1:I.Data.6;
   EMG_STOP_PB_LH : ALIAS FOR Local:2:I.Data.23;
   EXHAUST_SET_LIM : REAL := 0.5;
   EXHAUST_SET_STN1 : BOOL;
   EXHAUST_SET_STN2 : BOOL;
   EXHAUST_SET_STN3 : BOOL;
   EXHAUST_SET_STN4 : BOOL;
   EXHAUST_VALVE_STN1 : ALIAS FOR Local:1:O.Data.7;
   EXHAUST_VALVE_STN2 : ALIAS FOR Local:1:O.Data.15;
   EXHAUST_VALVE_STN3 : ALIAS FOR Local:3:O.Data.7;
   EXHAUST_VALVE_STN4 : ALIAS FOR Local:3:O.Data.15;
   EXHS_OFF_BLK_STN1 : FILL_VAL_OFF := (SET_SEQ_NO := 54, NEXT_SEQ_NO := 55);
   EXHS_OFF_BLK_STN2 : FILL_VAL_OFF := (SET_SEQ_NO := 54, NEXT_SEQ_NO := 55);
   EXHS_OFF_BLK_STN3 : FILL_VAL_OFF := (SET_SEQ_NO := 54, NEXT_SEQ_NO := 55);
   EXHS_OFF_BLK_STN4 : FILL_VAL_OFF := (SET_SEQ_NO := 54, NEXT_SEQ_NO := 55);
   EXHS_OK_DEL_STN3 : TIMER := (PRE := 500);
   EXHS_VAL_HP_ON_STN1 : BOOL;
   EXHS_VAL_HP_ON_STN3 : BOOL;
   EXHS_VAL_HP_ON_STN4 : BOOL;
   EXHS_VAL_OFF_CE_STN4 : BOOL;
   EXHS_VAL_OFF_CONS_STN2 : BOOL;
   EXHS_VAL_OFF_STN1 : BOOL;
   EXHS_VAL_OFF_STN2 : BOOL;
   EXHS_VAL_OFF_STN3 : BOOL;
   EXHS_VAL_OFF_STN4 : BOOL;
   EXHS_VAL_OFF_TE_STN4 : BOOL;
   EXHS_VAL_ON_STN1 : BOOL;
   EXHS_VAL_ON_STN2 : BOOL;
   EXHS_VAL_ON_STN3 : BOOL;
   EXHS_VAL_ON_STN4 : BOOL;
   FAIL_ARRAY : DINT[4];
   FAIL_BIN_DOOR_PROXY : ALIAS FOR Local:2:I.Data.29;
   FAIL_BIN_FULL_STN1 : BOOL;
   FAIL_BIN_FULL_STN2 : BOOL;
   FAIL_BIN_FULL_STN3 : BOOL;
   FAIL_BIN_FULL_STN4 : BOOL;
   FAIL_BIN_LOCK_DEL : TIMER := (PRE := 1000, ACC := 1004, EN := 1, DN := 1);
   FAIL_BIN_LOCK_PS : ALIAS FOR Local:2:I.Data.26;
   FAIL_BIN_SEL : BOOL;
   FAIL_BIN_SEQ_STN1 : INT;
   FAIL_BIN_SEQ_STN2 : INT;
   FAIL_BIN_SEQ_STN3 : INT;
   FAIL_BIN_SEQ_STN4 : INT;
   FAIL_BIN_UNLOCK_DOL : BOOL;
   FAIL_CLR_ONS_STN1 : BOOL;
   FAIL_CLR_ONS_STN2 : BOOL;
   FAIL_CLR_ONS_STN3 : BOOL;
   FAIL_CLR_ONS_STN4 : BOOL;
   FAIL_COMP_SENSOR : ALIAS FOR Local:2:I.Data.25;
   FAIL_COUNT_RETEST : DINT;
   FAIL_COUNT_RETEST_STN2 : DINT;
   FAIL_COUNT_STN1 : DINT;
   FAIL_COUNT_STN2 : DINT;
   FAIL_COUNT_STN3 : DINT := 1;
   FAIL_COUNT_STN4 : DINT;
   FAIL_COUNTER_RETEST : COUNTER := (PRE := 9999);
   FAIL_COUNTER_RETEST_STN2 : COUNTER := (PRE := 9999);
   FAIL_COUNTER_STN1 : COUNTER := (PRE := 9999);
   FAIL_COUNTER_STN2 : COUNTER := (PRE := 9999);
   FAIL_COUNTER_STN3 : COUNTER := (PRE := 9999, ACC := 1);
   FAIL_COUNTER_STN4 : COUNTER := (PRE := 9999);
   FAIL_FIFO_DEL : TIMER := (PRE := 250, ACC := 251);
   FAIL_FIFO_INDEX : DINT;
   FAIL_FIFO_STN1 : BOOL;
   FAIL_FIFO_STN2 : BOOL;
   FAIL_FIFO_STN3 : BOOL;
   FAIL_FIFO_STN4 : BOOL;
   FAIL_R1 : CONTROL := (LEN := 4, EM := 1);
   FAIL_RST_KS : ALIAS FOR Local:2:I.Data.14;
   FAIL_RST_ONS_STN1 : BOOL;
   FAIL_RST_ONS_STN2 : BOOL;
   FAIL_RST_ONS_STN3 : BOOL;
   FAIL_RST_ONS_STN4 : BOOL;
   FAILED_STN1 : BOOL;
   FAILED_STN2 : BOOL;
   FAILED_STN3 : BOOL;
   FAILED_STN4 : BOOL;
   FAULT_ARRAY : DINT[4];
   FAULT_BIN_DOOR_PROXY : ALIAS FOR Local:2:I.Data.30;
   FAULT_BIN_LOCK_DEL : TIMER := (PRE := 1000, ACC := 1004, EN := 1, DN := 1);
   FAULT_BIN_LOCK_PS : ALIAS FOR Local:2:I.Data.27;
   FAULT_BIN_SEL : BOOL;
   FAULT_BIN_UNLOCK_SOL : BOOL;
   FAULT_COUNT_STN1 : DINT;
   FAULT_COUNT_STN2 : DINT;
   FAULT_COUNT_STN3 : DINT := 2;
   FAULT_COUNT_STN4 : DINT;
   FAULT_COUNTER_STN1 : COUNTER := (PRE := 9999);
   FAULT_COUNTER_STN2 : COUNTER := (PRE := 9999);
   FAULT_COUNTER_STN3 : COUNTER := (PRE := 9999, ACC := 2);
   FAULT_COUNTER_STN4 : COUNTER := (PRE := 9999);
   FAULT_FIFO_STN1 : BOOL;
   FAULT_FIFO_STN2 : BOOL;
   FAULT_FIFO_STN3 : BOOL;
   FAULT_FIFO_STN4 : BOOL;
   FAULT_LAMP_STN1 : ALIAS FOR Local:3:O.Data.19;
   FAULT_LAMP_STN2 : ALIAS FOR Local:3:O.Data.23;
   FAULT_LAMP_STN3 : ALIAS FOR Local:3:O.Data.28;
   FAULT_LAMP_STN4 : ALIAS FOR REM:O.Data[0].0;
   FAULT_R1 : CONTROL := (LEN := 4, EM := 1);
   FAULTED_STN1 : BOOL;
   FAULTED_STN2 : BOOL;
   FAULTED_STN3 : BOOL;
   FAULTED_STN4 : BOOL;
   FILL_ACT_TIME_STN1 : REAL := 3.0;
   FILL_ACT_TIME_STN2 : REAL := 3.0;
   FILL_ACT_TIME_STN3 : REAL := 3.003;
   FILL_ACT_TIME_STN4 : REAL := 3.002;
   FILL_CHK_STN1 : PR_CHECK := (SET_SEQ := 30, ACT_PR := -0.05, PR_LL := 130.0, PR_HL := 145.0, SET_TIME := 3.0, ACT_TIME := 3.0, PR_AT_END := 141.43277, SEQ_STS_CODE := 4, RUN_CODE := 10, LIM_LOW_CODE := 18, LIM_HIGH_CODE := 19, NEXT_SEQ_NO := 35);
   FILL_CHK_STN2 : PR_CHECK := (SET_SEQ := 30, ACT_PR := -0.015992021, PR_LL := 130.0, PR_HL := 145.0, SET_TIME := 3.0, ACT_TIME := 3.0, PR_AT_END := 141.84927, SEQ_STS_CODE := 4, RUN_CODE := 10, LIM_LOW_CODE := 18, LIM_HIGH_CODE := 19, NEXT_SEQ_NO := 35);
   FILL_CHK_STN3 : PR_CHECK := (SET_SEQ := 30, PR_LL := 130.0, PR_HL := 145.0, SET_TIME := 3.0, ACT_TIME := 3.003, PR_AT_END := 141.75935, SEQ_STS_CODE := 4, RUN_CODE := 10, LIM_LOW_CODE := 18, LIM_HIGH_CODE := 19, NEXT_SEQ_NO := 35);
   FILL_CHK_STN4 : PR_CHECK := (SET_SEQ := 30, ACT_PR := 0.015994694, PR_LL := 130.0, PR_HL := 145.0, SET_TIME := 3.0, ACT_TIME := 3.002, PR_AT_END := 142.2088, SEQ_STS_CODE := 4, RUN_CODE := 10, LIM_LOW_CODE := 18, LIM_HIGH_CODE := 19, NEXT_SEQ_NO := 35);
   FILL_HIGH_STN1 : BOOL;
   FILL_HIGH_STN2 : BOOL;
   FILL_HIGH_STN3 : BOOL;
   FILL_HIGH_STN4 : BOOL;
   FILL_HL_STN1 : REAL := 145.0;
   FILL_HL_STN2 : REAL;
   FILL_HL_STN3 : REAL;
   FILL_HL_STN4 : REAL := 40.0;
   FILL_LL_STN1 : REAL := 130.0;
   FILL_LL_STN2 : REAL;
   FILL_LL_STN3 : REAL;
   FILL_LL_STN4 : REAL;
   FILL_LOW_STN1 : BOOL;
   FILL_LOW_STN2 : BOOL;
   FILL_LOW_STN3 : BOOL;
   FILL_LOW_STN4 : BOOL;
   FILL_SEQ_START_STN : SEQ_START_AND_FILL := (SET_SEQ_NO := 26, NEXT_SEQ_NO := 30);
   FILL_SEQ_START_STN2 : SEQ_START_AND_FILL := (SET_SEQ_NO := 26, NEXT_SEQ_NO := 30);
   FILL_SEQ_START_STN3 : SEQ_START_AND_FILL := (SET_SEQ_NO := 26, NEXT_SEQ_NO := 30);
   FILL_SEQ_START_STN4 : SEQ_START_AND_FILL := (SET_SEQ_NO := 26, NEXT_SEQ_NO := 30);
   FILL_SET_TIME : REAL := 3.0;
   FILL_VAL_OFF_SEQ_STN1 : FILL_VAL_OFF := (SET_SEQ_NO := 35, NEXT_SEQ_NO := 40);
   FILL_VAL_OFF_SEQ_STN2 : FILL_VAL_OFF := (SET_SEQ_NO := 35, NEXT_SEQ_NO := 40);
   FILL_VAL_OFF_SEQ_STN3 : FILL_VAL_OFF := (SET_SEQ_NO := 35, NEXT_SEQ_NO := 40);
   FILL_VAL_OFF_SEQ_STN4 : FILL_VAL_OFF := (SET_SEQ_NO := 35, NEXT_SEQ_NO := 40);
   FILL_VAL_OFF_STN1 : BOOL;
   FILL_VAL_OFF_STN2 : BOOL;
   FILL_VAL_OFF_STN3 : BOOL;
   FILL_VAL_OFF_STN4 : BOOL;
   FILL_VAL_ON_STN1 : BOOL;
   FILL_VAL_ON_STN2 : BOOL;
   FILL_VAL_ON_STN3 : BOOL := 1;
   FILL_VAL_ON_STN4 : BOOL;
   FINAL_PR_BOTTOM_CLAMP : BOOL;
   FINAL_PR_STN1 : BOOL;
   FINAL_PR_STN2 : BOOL;
   FINAL_PR_STN3 : BOOL;
   FINAL_PR_STN4 : BOOL;
   FINAL_PR_TOP_CLAMP : BOOL;
   FIX_DOWN_LS : BOOL;
   FIX_DOWN_SET : BOOL;
   FIX_UP_LS : BOOL;
   FIX_UP_SET : BOOL;
   FLT_CLR_ONS : BOOL;
   FLT_CLR_ONS_OP20A : DINT; {produced}
   FLT_CLR_ONS_OP20B : DINT; {produced}
   FLT_CLR_ONS_OP20C : DINT; {produced}
   FLT_CLR_ONS_OP20D : DINT; {produced}
   FLT_CLR_ONS_STN1 : BOOL;
   FLT_CLR_ONS_STN2 : BOOL;
   FLT_CLR_ONS_STN3 : BOOL;
   FLT_CLR_ONS_STN4 : BOOL;
   FLT_CODE_STN1 : DINT;
   FLT_CODE_STN2 : DINT;
   FLT_CODE_STN3 : DINT;
   FLT_CODE_STN4 : DINT := 18;
   FLT_RST_PB_STN1 : ALIAS FOR Local:1:I.Data.7;
   FLT_RST_PB_STN2 : ALIAS FOR Local:1:I.Data.8;
   FLT_RST_PB_STN3 : ALIAS FOR Local:1:I.Data.9;
   FLT_RST_PB_STN4 : ALIAS FOR Local:2:I.Data.15;
   FP_ACCESS_OK : ALIAS FOR Local:2:I.Data.24;
   GET_FIRST_FAILED : DINT;
        .1   // STN2 FAILED
        .2   // STN3 FAILED
        .3   // STN4 FAILED
        .0   // STN1 FAILED
   GOTO_FAIL_BIN_STN2 : DINT;
   GOTO_FAIL_BIN_STN3 : DINT;
   GOTO_FAIL_BIN_STN4 : DINT;
   GOTO_FAULT_BIN_STN1 : DINT;
   GOTO_FAULT_BIN_STN2 : DINT;
   HIDE_MAIN_MENU : BOOL;
   HOME_COND_NOK_STN1 : BOOL;
   HOME_COND_NOK_STN2 : BOOL;
   HOME_COND_NOK_STN3 : BOOL;
   HOME_COND_NOK_STN4 : BOOL;
   HOME_COND_OK_STN1 : BOOL := 1;
   HOME_COND_OK_STN2 : BOOL := 1;
   HOME_COND_OK_STN3 : BOOL := 1;
   HOME_COND_OK_STN4 : BOOL := 1;
   HP_ACT_DROP_STN1 : REAL := 0.49569702;
   HP_ACT_DROP_STN2 : REAL := 0.5277252;
   HP_ACT_DROP_STN3 : REAL := 0.5121765;
   HP_ACT_DROP_STN4 : REAL := 0.4958496; {produced}
   HP_ACT_PR_STN1 : REAL := -0.05;
   HP_ACT_PR_STN2 : REAL := -0.015992021;
   HP_ACT_PR_STN3 : REAL;
   HP_ACT_PR_STN4 : REAL; {produced}
   HP_FILL_VALVE_SET_STN1 : BOOL;
   HP_FILL_VALVE_SET_STN2 : BOOL;
   HP_FILL_VALVE_SET_STN3 : BOOL;
   HP_FILL_VALVE_SET_STN4 : BOOL;
   HP_FILL_VALVE_STN1 : ALIAS FOR Local:1:O.Data.8;
   HP_FILL_VALVE_STN2 : ALIAS FOR Local:3:O.Data.0;
   HP_FILL_VALVE_STN3 : ALIAS FOR Local:3:O.Data.8;
   HP_FILL_VALVE_STN4 : ALIAS FOR Local:3:O.Data.16;
   HP_P2_STN1 : REAL := 138.5545;
   HP_P2_STN2 : REAL := 138.89075;
   HP_P2_STN3 : REAL := 138.6063;
   HP_P2_STN4 : REAL := 139.29776;
   HP_RESULT : DINT := 5; {produced}
   HP_RESULT_STN1 : DINT := 2;
   HP_RESULT_STN2 : DINT := 2;
   HP_RESULT_STN3 : DINT := 2;
   HP_RESULT_STN4 : DINT := 2;
   HP_SENSOR_SEL : BOOL;
   HP_STS_STN1 : DINT := 2;
   HP_STS_STN2 : DINT := 2;
   HP_STS_STN3 : DINT := 2;
   HP_STS_STN4 : DINT := 2;
   HP_TEST_ON : BOOL := 1;
   INCORRECT_STN1 : BOOL;
   INCORRECT_STN2 : BOOL;
   INCORRECT_STN3 : BOOL;
   INCORRECT_STN4 : BOOL;
   INDV_CT_OFF_STN1 : BOOL;
   INDV_CT_OFF_STN2 : BOOL;
   INDV_CT_OFF_STN3 : BOOL;
   INDV_CT_OFF_STN4 : BOOL;
   INDV_CTEST_ON_STN1 : BOOL;
   INDV_CTEST_ON_STN2 : BOOL;
   INDV_CTEST_ON_STN3 : BOOL;
   INDV_CTEST_ON_STN4 : BOOL;
   INDV_CTEST_SEL_STN1 : BOOL;
   INDV_CTEST_SEL_STN2 : BOOL;
   INDV_CTEST_SEL_STN3 : BOOL;
   INDV_CTEST_SEL_STN4 : BOOL;
   INDV_LT_OFF_STN1 : BOOL;
   INDV_LT_OFF_STN2 : BOOL;
   INDV_LT_OFF_STN3 : BOOL;
   INDV_LT_OFF_STN4 : BOOL;
   INDV_LTEST_SEL_STN1 : BOOL;
   INDV_LTEST_SEL_STN2 : BOOL;
   INDV_LTEST_SEL_STN3 : BOOL;
   INDV_LTEST_SEL_STN4 : BOOL;
   INDV_TEST_ON_STN1 : BOOL;
   INDV_TEST_ON_STN2 : BOOL;
   INDV_TEST_ON_STN3 : BOOL;
   INDV_TEST_ON_STN4 : BOOL;
   INIT_STN1 : BOOL;
   INIT_STN2 : BOOL;
   INIT_STN3 : BOOL;
   INIT_STN4 : BOOL;
   INITIAL_PR_BOTTOM_CLAMP : BOOL;
   INITIAL_PR_STN1 : BOOL;
   INITIAL_PR_STN2 : BOOL;
   INITIAL_PR_STN3 : BOOL;
   INITIAL_PR_STN4 : BOOL;
   INITIAL_PR_TOP_CLAMP : BOOL;
   INLET_AIR_DPS : ALIAS FOR Local:1:I.Data.0;
   INLET_AIR_HPS : ALIAS FOR Local:1:I.Data.1;
   INLET_AIR_LOW : TIMER := (PRE := 3000);
   INLET_AIR_SOL : ALIAS FOR Local:1:O.Data.0;
   INPUT_1_16 : INT := -31677;
   LH_START_PB_STN1 : ALIAS FOR Local:1:I.Data.2;
   LH_START_PB_STN2 : ALIAS FOR Local:1:I.Data.3;
   LH_START_PB_STN3 : ALIAS FOR Local:1:I.Data.4;
   LH_START_PB_STN4 : ALIAS FOR Local:1:I.Data.5;
   LOCK_FAIL_BIN : BOOL;
   LOGIN_LEVEL : INT;
   LT_COMPLETED_STN1 : BOOL := 1;
   LT_COMPLETED_STN2 : BOOL := 1;
   LT_COMPLETED_STN3 : BOOL := 1;
   LT_COMPLETED_STN4 : BOOL := 1;
   LT_P1_STN1 : REAL := 141.43277;
   LT_P1_STN2 : REAL := 141.84927;
   LT_P1_STN3 : REAL := 141.75935;
   LT_P1_STN4 : REAL := 142.2088;
   LT_POKEYOKE_STN1 : DINT;
   LT_POKEYOKE_STN2 : DINT;
   LT_POKEYOKE_STN3 : DINT;
   LT_POKEYOKE_STN4 : DINT;
   MAIN_MENU : BOOL;
   MAIN_MENU_OFF : TIMER := (PRE := 150);
   MASTER_PR : REAL := 3000.942;
   MASTER_PR_CONS : REAL := 3000.942;
   MASTER_PR_SCL : SCP := (Y := 3000.942, X := 3.031, X1 := 0.575, X2 := 2.503, Y1 := 508.0, Y2 := 2465.0);
   MASTER_WORK_MAIN_MENU_EN : BOOL := 1;
   MODEL_SELECTED : STRING := '29047345';
   MOTOR_DOWN : ALIAS FOR REM:O.Data[1].3;
   MOTOR_RUN_STS : BOOL;
   MOTOR_SAFETY : BOOL := 1;
   MOTOR_UP : ALIAS FOR REM:O.Data[1].2;
   MPCB_TRIP : BOOL;
   MSB_EIP_1_16 : INT;
   MSG_STN1 : DINT := 1;
   MSG_STN2 : DINT := 1;
   MSG_STN3 : DINT := 1;
   MSG_STN4 : DINT := 1;
   NEXT_SEQ_NO_STN1 : DINT;
   NO_COMP_FAULT_STN1 : BOOL := 1;
   NO_COMP_FAULT_STN2 : BOOL := 1;
   NO_COMP_FAULT_STN3 : BOOL := 1;
   NO_COMP_FAULT_STN4 : BOOL := 1;
   NO_SYSTEM_FAULT_STN1 : BOOL := 1;
   NO_SYSTEM_FAULT_STN2 : BOOL := 1;
   NO_SYSTEM_FAULT_STN3 : BOOL := 1;
   NO_SYSTEM_FAULT_STN4 : BOOL := 1;
   NOT_FAILED_STN1 : BOOL := 1;
   NOT_FAILED_STN2 : BOOL := 1;
   NOT_FAILED_STN3 : BOOL := 1;
   NOT_FAILED_STN4 : BOOL := 1;
   ONS34 : BOOL;
   ONS5 : BOOL;
   OTHER_CAL_EDIT_MODE : BOOL;
   OTHER_CAL_VIEW_MODE : BOOL;
   OTHER_SENSOR_SEL : BOOL;
   P1_STN1 : REAL;
   P1_STN2 : REAL;
   P1_STN3 : REAL;
   P1_STN4 : REAL;
   P2_STN1 : REAL := 139.0502;
   P2_STN2 : REAL := 139.41847;
   P2_STN3 : REAL := 139.11847;
   P2_STN4 : REAL := 139.79361;
   PASS_BIN_COUNT : DINT := 100;
   PASS_BIN_FULL : DINT;
   PASS_COUNT_RETEST : DINT;
   PASS_COUNT_RETEST_STN2 : DINT;
   PASS_COUNT_STN1 : DINT := 4;
   PASS_COUNT_STN2 : DINT := 9;
   PASS_COUNT_STN3 : DINT := 12;
   PASS_COUNT_STN4 : DINT;
   PASS_COUNTER_RETEST : COUNTER := (PRE := 9999);
   PASS_COUNTER_RETEST_STN2 : COUNTER := (PRE := 9999);
   PASS_LAMP_STN1 : ALIAS FOR Local:3:O.Data.18;
   PASS_LAMP_STN2 : ALIAS FOR Local:3:O.Data.22;
   PASS_LAMP_STN3 : ALIAS FOR Local:3:O.Data.27;
   PASS_LAMP_STN4 : ALIAS FOR Local:3:O.Data.31;
   PASSED_STN1 : BOOL := 1;
   PASSED_STN2 : BOOL := 1;
   PASSED_STN3 : BOOL := 1;
   PASSED_STN4 : BOOL := 1;
   PASSWORD_SET : DINT;
   PLC_LIVE_BIT : BOOL;
   POKEYOKE_NOT_DONE : BOOL;
   PR_C_MASTER : REAL;
   PR_C_STAMP : REAL;
   PR_C_STN1 : REAL;
   PR_C_STN2 : REAL;
   PR_C_STN3 : REAL;
   PR_C_STN4 : REAL;
   PR_C_WORK : REAL;
   PR_DIFF_ACT_STN1 : REAL := 73.106445;
   PR_DIFF_ACT_STN2 : REAL := 102.48828;
   PR_DIFF_ACT_STN3 : REAL := 129.26184;
   PR_DIFF_ACT_STN4 : REAL := 80.18457;
   PR_DIFF_CALB_ACT : REAL := 323.9121;
   PR_DIFF_HL : REAL := 500.0;
   PR_DIFF_LL : REAL := 50.0;
   PR_DIFF_SET : REAL;
   PR_DIFF_TARRED_STN1 : REAL := -498.3689;
   PR_DIFF_TARRED_STN2 : REAL := -469.7915;
   PR_DIFF_TARRED_STN3 : REAL := -483.83057;
   PR_DIFF_TARRED_STN4 : REAL := -478.98828;
   PR_DIFF_TEST_ACT_STN1 : REAL := 2174.0005;
   PR_DIFF_TEST_ACT_STN2 : REAL := 2160.7444;
   PR_DIFF_TEST_ACT_STN3 : REAL := 465.65845;
   PR_DIFF_TEST_ACT_STN4 : DINT := 24;
   PR_EXHS_LIM : REAL := 0.5;
   PR_EXHS_OK_STN1 : BOOL;
   PR_EXHS_OK_STN2 : BOOL;
   PR_EXHS_OK_STN3 : BOOL;
   PR_EXHS_OK_STN4 : BOOL;
   PR_SCL_STN1 : SCP := (Y := -0.05, X := -0.001, X1 := -0.001, X2 := 9.758, Y1 := -0.05, Y2 := 156.0);
   PR_SCL_STN2 : SCP := (Y := -0.015992021, X := -0.005, X1 := -0.004, X2 := 9.779, Y2 := 156.45);
   PR_SCL_STN3 : SCP := (X2 := 9.728, Y2 := 155.7);
   PR_SCL_STN4 : SCP := (X := -0.004, X1 := -0.004, X2 := 9.793, Y2 := 156.7);
   PR_X1_MASTER : REAL := 0.575;
   PR_X1_STAMP : REAL;
   PR_X1_STN1 : REAL := -0.001;
   PR_X1_STN2 : REAL := -0.004;
   PR_X1_STN3 : REAL;
   PR_X1_STN4 : REAL := -0.004;
   PR_X1_WORK : REAL := 1.999;
   PR_X2_MASTER : REAL := 2.503;
   PR_X2_STAMP : REAL := 5.798;
   PR_X2_STN1 : REAL := 9.758;
   PR_X2_STN2 : REAL := 9.779;
   PR_X2_STN3 : REAL := 9.728;
   PR_X2_STN4 : REAL := 9.793;
   PR_X2_WORK : REAL := 9.669;
   PR_X_MASTER : REAL := 3.031;
   PR_X_STAMP : REAL := 4.552;
   PR_X_STN1 : REAL := -0.001;
   PR_X_STN2 : REAL := -0.005;
   PR_X_STN3 : REAL;
   PR_X_STN4 : REAL := -0.004;
   PR_X_WORK : REAL := 10.5;
   PR_Y1_MASTER : REAL := 508.0;
   PR_Y1_STAMP : REAL;
   PR_Y1_STN1 : REAL := -0.05;
   PR_Y1_STN2 : REAL;
   PR_Y1_STN3 : REAL;
   PR_Y1_STN4 : REAL;
   PR_Y1_WORK : REAL := 508.0;
   PR_Y2_MASTER : REAL := 2465.0;
   PR_Y2_STAMP : REAL := 5.799;
   PR_Y2_STN1 : REAL := 156.0;
   PR_Y2_STN2 : REAL := 156.45;
   PR_Y2_STN3 : REAL := 155.7;
   PR_Y2_STN4 : REAL := 156.7;
   PR_Y2_WORK : REAL := 2465.0;
   PYOKE_LT_STN1 : BOOL;
   PYOKE_LT_STN2 : BOOL;
   PYOKE_LT_STN3 : BOOL;
   PYOKE_LT_STN4 : BOOL;
   RESET_COUNT_RETEST : BOOL;
   RESET_COUNT_RETEST_STN2 : BOOL;
   RESET_COUNT_STN1 : BOOL;
   RESET_COUNT_STN2 : BOOL;
   RESET_COUNT_STN3 : BOOL;
   RESET_COUNT_STN4 : BOOL;
   RESET_SEQ_BLK_STN1 : Rst_Seq_On := (INPUT_1_16 := 1088, PR_EXHS_LIMIT := 0.5);
   RESET_SEQ_BLK_STN2 : Rst_Seq_On := (INPUT_1_16 := 1088, PR_EXHS_LIMIT := 0.5);
   RESET_SEQ_BLK_STN3 : Rst_Seq_On := (INPUT_1_16 := 1088, PR_EXHS_LIMIT := 0.5);
   RESET_SEQ_BLK_STN4 : Rst_Seq_On := (INPUT_1_16 := 1088, PR_EXHS_LIMIT := 0.5);
   RESET_SEQ_STN3 : Rst_Seq_On;
   RESET_SEQ_STN4 : Rst_Seq_On;
   RETEST : BOOL;
   RETEST_FAIL_COUNT : DINT;
   RETEST_ON_PROHIBIT : BOOL;
   RETEST_PASS_COUNT : DINT;
   RETEST_SET_COUNT : DINT;
   RFID_STN1 : STRING;
   RFID_STN2 : STRING;
   RFID_STN3 : STRING;
   RFID_STN4 : STRING := '0029047345L0721Gj000013';
   RH_START_PB_STN1 : BOOL;
   RH_START_PB_STN2 : BOOL;
   RH_START_PB_STN3 : BOOL;
   RH_START_PB_STN4 : BOOL;
   RST_BOTTOM_DECLAMP_OK_STN1 : BOOL;
   RST_BOTTOM_DECLAMP_OK_STN3 : BOOL;
   RST_BOTTOM_DECLAMP_OK_STN4 : BOOL;
   RST_BOTTOM_DECLAMP_STN1 : BOOL;
   RST_BOTTOM_DECLAMP_STN2 : BOOL;
   RST_BOTTOM_DECLAMP_STN3 : BOOL;
   RST_BOTTOM_DECLAMP_STN4 : BOOL;
   RST_DOOR_NOT_OPEN_STN1 : BOOL;
   RST_DOOR_NOT_OPENED_STN4 : BOOL;
   RST_DOOR_OPEN_BLK_STN1 : DA_SOL_FWD_SEQ := (DA_SOL_PS := 1, RUN_CODE := 3, FLT_CODE := 27, NEXT_SEQ_NO := 118);
   RST_DOOR_OPEN_BLK_STN2 : DA_SOL_FWD_SEQ := (DA_SOL_PS := 1, RUN_CODE := 3, FLT_CODE := 27, NEXT_SEQ_NO := 118);
   RST_DOOR_OPEN_BLK_STN3 : DA_SOL_FWD_SEQ := (DA_SOL_PS := 1, RUN_CODE := 3, FLT_CODE := 27, NEXT_SEQ_NO := 118);
   RST_DOOR_OPEN_BLK_STN4 : DA_SOL_FWD_SEQ := (DA_SOL_PS := 1, RUN_CODE := 3, FLT_CODE := 27, NEXT_SEQ_NO := 118);
   RST_DOOR_OPEN_ON : BOOL;
   RST_DOOR_OPEN_ON_STN2 : BOOL;
   RST_DOOR_OPEN_ON_STN3 : BOOL;
   RST_DOOR_OPEN_ON_STN4 : BOOL;
   RST_DOOR_OPEN_SEQ : DINT;
   RST_DOOR_OPEN_SEQ_STN2 : DINT;
   RST_DOOR_OPEN_SEQ_STN3 : DINT;
   RST_DOOR_OPEN_SEQ_STN4 : DINT;
   RST_DOOR_OPEN_STN1 : BOOL;
   RST_DOOR_OPEN_STN2 : BOOL;
   RST_DOOR_OPEN_STN3 : BOOL;
   RST_DOOR_OPEN_STN4 : BOOL;
   RST_EXHS_VAL_OFF_STN1 : BOOL;
   RST_EXHS_VAL_OFF_STN2 : BOOL;
   RST_EXHS_VAL_OFF_STN3 : BOOL;
   RST_EXHS_VAL_OFF_STN4 : BOOL;
   RST_FLT_CLR_ONS_STN1 : BOOL;
   RST_SEQ_ON_STN1 : BOOL;
   RST_SEQ_ON_STN2 : BOOL;
   RST_SEQ_ON_STN3 : BOOL;
   RST_SEQ_ON_STN4 : BOOL;
   RST_SEQ_OVER_STN1 : BOOL;
   RST_SEQ_OVER_STN2 : BOOL;
   RST_SEQ_OVER_STN3 : BOOL;
   RST_SEQ_OVER_STN4 : BOOL;
   RST_TEST_VAL_OFF_STN1 : BOOL;
   RST_TEST_VAL_OFF_STN2 : BOOL;
   RST_TEST_VAL_OFF_STN3 : BOOL;
   RST_TEST_VAL_OFF_STN4 : BOOL;
   RST_TOP_DECLAMP_AUTO_STN1 : BOOL;
   RST_TOP_DECLAMP_AUTO_STN2 : BOOL;
   RST_TOP_DECLAMP_AUTO_STN3 : BOOL;
   RST_TOP_DECLAMP_AUTO_STN4 : BOOL;
   RST_TOP_DECLAMP_OK_STN1 : BOOL;
   RST_TOP_DECLAMP_OK_STN2 : BOOL;
   RST_TOP_DECLAMP_OK_STN3 : BOOL;
   RST_TOP_DECLAMP_OK_STN4 : BOOL;
   RST_TOP_DECLAMP_STN1 : BOOL;
   RST_TOP_DECLAMP_STN2 : BOOL;
   RST_TOP_DECLAMP_STN3 : BOOL;
   RST_TOP_DECLAMP_STN4 : BOOL;
   RUN_CODE_STN1 : DINT;
   SCAN_OK_STN1 : BOOL;
   SCAN_OK_STN2 : BOOL;
   SCAN_OK_STN3 : BOOL;
   SCAN_OK_STN4 : BOOL;
   SCR_STS : DINT[6] := ([1] := 11, [2] := 1, [3] := 1, [4] := 1, [5] := 1);
   SENS_CAL_EDIT_MODE : BOOL;
   SENS_CAL_SEL_BOTTOM_CLAMP : BOOL;
   SENS_CAL_SEL_MASTER : BOOL;
   SENS_CAL_SEL_STAMP : BOOL;
   SENS_CAL_SEL_TOP_CLAMP : BOOL;
   SENS_CAL_VIEW_MODE : BOOL;
   SENS_CALB_SEL_STN1 : BOOL;
   SENS_CALB_SEL_STN2 : BOOL;
   SENS_CALB_SEL_STN3 : BOOL;
   SENS_CALB_SEL_STN4 : BOOL;
   SEQ_NO_STN1 : DINT := 1;
   SEQ_NO_STN2 : DINT := 1;
   SEQ_NO_STN3 : DINT := 1;
   SEQ_NO_STN4 : DINT := 120;
   SET_240 : REAL := 144000.0;
   SET_DISTANCE : REAL := 600.0;
   SET_DROP : REAL := 1.0;
   SET_MENU_STN1_EN : BOOL := 1;
   SET_MENU_STN2_EN : BOOL := 1;
   SET_MENU_STN3_EN : BOOL := 1;
   SET_MENU_STN4_EN : BOOL := 1;
   SET_MODE_SEL_STN1 : BOOL;
   SET_MODE_SEL_STN2 : BOOL;
   SET_MODE_SEL_STN3 : BOOL;
   SET_MODE_SEL_STN4 : BOOL;
   SET_TIMER : REAL := 183439.48;
   SET_TRAVEL : REAL := 785.0;
   SLIDE_TRAVEL : TIMER := (PRE := 183439, ACC := 2808834);
   STAB_ACT_TIME_STN1 : REAL := 5.002;
   STAB_ACT_TIME_STN2 : REAL := 5.0;
   STAB_ACT_TIME_STN3 : REAL := 5.001;
   STAB_ACT_TIME_STN4 : REAL := 5.0;
   STAB_CHK_STN1 : PR_CHECK := (SET_SEQ := 40, ACT_PR := -0.05, PR_LL := 130.0, PR_HL := 145.0, SET_TIME := 5.0, ACT_TIME := 5.002, PR_AT_END := 139.0502, SEQ_STS_CODE := 4, RUN_CODE := 12, LIM_LOW_CODE := 20, LIM_HIGH_CODE := 21, NEXT_SEQ_NO := 45);
   STAB_CHK_STN2 : PR_CHECK := (SET_SEQ := 40, ACT_PR := -0.015992021, PR_LL := 130.0, PR_HL := 145.0, SET_TIME := 5.0, ACT_TIME := 5.0, PR_AT_END := 139.41847, SEQ_STS_CODE := 4, RUN_CODE := 12, LIM_LOW_CODE := 20, LIM_HIGH_CODE := 21, NEXT_SEQ_NO := 45);
   STAB_CHK_STN3 : PR_CHECK := (SET_SEQ := 40, ACT_PR := 0.016005347, PR_LL := 130.0, PR_HL := 145.0, SET_TIME := 5.0, ACT_TIME := 5.001, PR_AT_END := 139.11847, SEQ_STS_CODE := 4, RUN_CODE := 12, LIM_LOW_CODE := 20, LIM_HIGH_CODE := 21, NEXT_SEQ_NO := 45);
   STAB_CHK_STN4 : PR_CHECK := (SET_SEQ := 40, PR_LL := 130.0, PR_HL := 145.0, SET_TIME := 5.0, ACT_TIME := 5.0, PR_AT_END := 139.79361, SEQ_STS_CODE := 4, RUN_CODE := 12, LIM_LOW_CODE := 20, LIM_HIGH_CODE := 20, NEXT_SEQ_NO := 45);
   STAB_HIGH_STN1 : BOOL;
   STAB_HIGH_STN2 : BOOL;
   STAB_HIGH_STN3 : BOOL;
   STAB_HIGH_STN4 : BOOL;
   STAB_LOW_STN1 : BOOL;
   STAB_LOW_STN2 : BOOL;
   STAB_LOW_STN3 : BOOL;
   STAB_LOW_STN4 : BOOL;
   STAB_SET_TIME : REAL := 5.0;
   STAMP_BLK_STN1 : STAMP_SEQ := (SET_SEQ_NO := 85, STAMP_RET_OK := 1, FLT_CODE := 36, RUN_CODE := 21, NEXT_SEQ_NO := 90);
   STAMP_BLK_STN2 : STAMP_SEQ := (SET_SEQ_NO := 85, STAMP_RET_OK := 1, FLT_CODE := 36, RUN_CODE := 21, NEXT_SEQ_NO := 90);
   STAMP_BLK_STN3 : STAMP_SEQ := (SET_SEQ_NO := 85, STAMP_RET_OK := 1, FLT_CODE := 36, RUN_CODE := 21, NEXT_SEQ_NO := 90);
   STAMP_BLK_STN4 : STAMP_SEQ := (SET_SEQ_NO := 85, STAMP_RET_OK := 1, FLT_CODE := 36, RUN_CODE := 21, NEXT_SEQ_NO := 90);
   STAMP_FWD_OK_STN1 : BOOL;
   STAMP_FWD_OK_STN2 : BOOL;
   STAMP_FWD_OK_STN3 : BOOL;
   STAMP_FWD_OK_STN4 : BOOL;
   STAMP_HL : REAL := 5.0;
   STAMP_LL : REAL := 1.0;
   STAMP_NOT_FWD : BOOL;
   STAMP_NOT_FWD_STN2 : BOOL;
   STAMP_NOT_FWD_STN3 : BOOL;
   STAMP_NOT_FWD_STN4 : BOOL;
   STAMP_NOT_RET : BOOL;
   STAMP_NOT_RET_STN2 : BOOL;
   STAMP_NOT_RET_STN3 : BOOL;
   STAMP_NOT_RET_STN4 : BOOL;
   STAMP_ON_STN1 : BOOL;
   STAMP_ON_STN2 : BOOL;
   STAMP_ON_STN3 : BOOL;
   STAMP_ON_STN4 : BOOL;
   STAMP_PR : REAL := 4.551785;
   STAMP_PR_CHECK : TIMER := (PRE := 1000);
   STAMP_PR_DEL : TIMER := (PRE := 6000);
   STAMP_PR_HIGH_STN1 : BOOL;
   STAMP_PR_HIGH_STN2 : BOOL;
   STAMP_PR_HIGH_STN3 : BOOL;
   STAMP_PR_HIGH_STN4 : BOOL;
   STAMP_PR_LOW_STN1 : BOOL;
   STAMP_PR_LOW_STN2 : BOOL;
   STAMP_PR_LOW_STN3 : BOOL;
   STAMP_PR_LOW_STN4 : BOOL;
   STAMP_PR_SCL : SCP := (Y := 4.5527854, X := 4.552, X2 := 5.798, Y2 := 5.799);
   STAMP_PS_STN1 : ALIAS FOR Local:1:I.Data.14;
   STAMP_PS_STN2 : ALIAS FOR Local:2:I.Data.3;
   STAMP_PS_STN3 : ALIAS FOR Local:2:I.Data.8;
   STAMP_PS_STN4 : ALIAS FOR Local:2:I.Data.13;
   STAMP_SOL_STN1 : ALIAS FOR Local:1:O.Data.5;
   STAMP_SOL_STN2 : ALIAS FOR Local:1:O.Data.13;
   STAMP_SOL_STN3 : ALIAS FOR Local:3:O.Data.5;
   STAMP_SOL_STN4 : ALIAS FOR Local:3:O.Data.13;
   START_PB_ONS_STN1 : BOOL;
   START_PB_ONS_STN2 : BOOL;
   START_PB_ONS_STN3 : BOOL;
   START_PB_ONS_STN4 : BOOL;
   STN1_DB_SAVED : DINT;
   STN1_INPUT : INT;
   STN1_ON : BOOL := 1;
   STN1_TEST_STS : DINT := 2; {produced}
   STN1_TRACE_ON_STS : DINT := 1;
   STN2_DB_SAVED : DINT;
   STN2_ON : BOOL := 1;
   STN2_TEST_STS : DINT := 2; {produced}
   STN2_TRACE_ON_STS : DINT := 1;
   STN3_DB_SAVED : DINT;
   STN3_ON : BOOL := 1;
   STN3_TEST_STS : DINT := 2; {produced}
   STN3_TRACE_ON_STS : DINT := 1;
   STN4_DB_SAVED : DINT;
   STN4_ON : BOOL := 1;
   STN4_TEST_STS : DINT := 2; {produced}
   STN4_TRACE_ON_STS : DINT := 1;
   STOP_MOTOR : BOOL;
   STS : DINT := 13;
   STS_OP_STN1 : DINT;
   STS_OP_STN2 : DINT := 1;
   STS_OP_STN3 : DINT := 1;
   STS_OP_STN4 : DINT := 1;
   STS_STN1 : DINT;
   SYSTEM_FAULT_STN1 : BOOL;
   SYSTEM_FAULT_STN2 : BOOL;
   SYSTEM_FAULT_STN3 : BOOL;
   SYSTEM_FAULT_STN4 : BOOL;
   TARRED_CONS_VALUE : REAL;
   TARRED_VALUE_STN1 : REAL := 821.26587;
   TARRED_VALUE_STN2 : REAL := 793.7036;
   TARRED_VALUE_STN3 : REAL := 807.7427;
   TARRED_VALUE_STN4 : REAL := 802.9004;
   TEST_ACT_TIME_STN1 : REAL := 15.001;
   TEST_ACT_TIME_STN2 : REAL := 15.001;
   TEST_ACT_TIME_STN3 : REAL := 15.003;
   TEST_ACT_TIME_STN4 : REAL := 15.003;
   TEST_INIT_DEL : TIMER := (PRE := 250);
   TEST_INIT_DEL_STN1 : TIMER := (PRE := 250);
   TEST_LAMP_STN1 : ALIAS FOR Local:3:O.Data.17;
   TEST_LAMP_STN2 : ALIAS FOR Local:3:O.Data.21;
   TEST_LAMP_STN3 : ALIAS FOR Local:3:O.Data.26;
   TEST_LAMP_STN4 : ALIAS FOR Local:3:O.Data.30;
   TEST_ON_STN1 : BOOL;
   TEST_ON_STN2 : BOOL;
   TEST_ON_STN3 : BOOL;
   TEST_ON_STN4 : BOOL;
   TEST_OVER_DEL : TIMER := (PRE := 500);
   TEST_OVER_DEL_STN2 : TIMER := (PRE := 500);
   TEST_OVER_DEL_STN3 : TIMER := (PRE := 500);
   TEST_OVER_DEL_STN4 : TIMER := (PRE := 500);
   TEST_SET_TIME : REAL := 15.0;
   TEST_SOL_STN1 : ALIAS FOR Local:1:O.Data.6;
   TEST_SOL_STN2 : ALIAS FOR Local:1:O.Data.14;
   TEST_SOL_STN3 : ALIAS FOR Local:3:O.Data.6;
   TEST_SOL_STN4 : ALIAS FOR Local:3:O.Data.14;
   TEST_STS_STN1 : DINT := 1;
   TEST_STS_STN2 : DINT := 1;
   TEST_STS_STN3 : DINT := 1;
   TEST_STS_STN4 : DINT := 1;
   TEST_STS_UPDATE_STN1 : TEST_TAIL_END := (SET_SEQ_NO := 50, STN_ON := 1, LT_COMPLETED := 1, NEXT_SEQ_NO := 54);
   TEST_STS_UPDATE_STN2 : TEST_TAIL_END := (SET_SEQ_NO := 50, STN_ON := 1, LT_COMPLETED := 1, NEXT_SEQ_NO := 54);
   TEST_STS_UPDATE_STN3 : TEST_TAIL_END := (SET_SEQ_NO := 50, STN_ON := 1, LT_COMPLETED := 1, NEXT_SEQ_NO := 54);
   TEST_STS_UPDATE_STN4 : TEST_TAIL_END := (SET_SEQ_NO := 50, STN_ON := 1, LT_COMPLETED := 1, NEXT_SEQ_NO := 54);
   TEST_VAL_OFF_STN1 : BOOL;
   TEST_VAL_OFF_STN2 : BOOL;
   TEST_VAL_OFF_STN3 : BOOL;
   TEST_VAL_OFF_STN4 : BOOL;
   TEST_VAL_ON_STN1 : BOOL;
   TEST_VAL_ON_STN2 : BOOL;
   TEST_VAL_ON_STN3 : BOOL;
   TEST_VAL_ON_STN4 : BOOL;
   TEST_VALVE_STN1 : ALIAS FOR Local:1:O.Data.6;
   TIMER1_SET_VAL : DINT := 31;
   TIMER1_SET_VALUE : REAL := 183.43948;
   TOP_CLAMP_2BPR_HIGH : BOOL;
   TOP_CLAMP_2BPR_HIGH_STN2 : BOOL;
   TOP_CLAMP_2BPR_HIGH_STN3 : BOOL;
   TOP_CLAMP_2BPR_HIGH_STN4 : BOOL;
   TOP_CLAMP_2BPR_LOW : BOOL;
   TOP_CLAMP_2BPR_LOW_STN2 : BOOL;
   TOP_CLAMP_2BPR_LOW_STN3 : BOOL;
   TOP_CLAMP_2BPR_LOW_STN4 : BOOL;
   TOP_CLAMP_4BPR_HIGH : BOOL;
   TOP_CLAMP_4BPR_HIGH_STN2 : BOOL;
   TOP_CLAMP_4BPR_HIGH_STN3 : BOOL;
   TOP_CLAMP_4BPR_HIGH_STN4 : BOOL;
   TOP_CLAMP_4BPR_LOW : BOOL;
   TOP_CLAMP_4BPR_LOW_STN2 : BOOL;
   TOP_CLAMP_4BPR_LOW_STN3 : BOOL;
   TOP_CLAMP_4BPR_LOW_STN4 : BOOL;
   TOP_CLAMP_AUTO_STN1 : BOOL;
   TOP_CLAMP_AUTO_STN2 : BOOL;
   TOP_CLAMP_AUTO_STN3 : BOOL;
   TOP_CLAMP_AUTO_STN4 : BOOL;
   TOP_CLAMP_BLK_STN1 : DA_SOL_FWD_SEQ := (RUN_CODE := 4, FLT_CODE := 6, NEXT_SEQ_NO := 15);
   TOP_CLAMP_BLK_STN2 : DA_SOL_FWD_SEQ := (RUN_CODE := 4, FLT_CODE := 6, NEXT_SEQ_NO := 15);
   TOP_CLAMP_BLK_STN3 : DA_SOL_FWD_SEQ := (RUN_CODE := 4, FLT_CODE := 6, NEXT_SEQ_NO := 15);
   TOP_CLAMP_BLK_STN4 : DA_SOL_FWD_SEQ := (RUN_CODE := 4, FLT_CODE := 6, NEXT_SEQ_NO := 15);
   TOP_CLAMP_C : REAL;
   TOP_CLAMP_FAULT_STN1 : BOOL;
   TOP_CLAMP_FAULT_STN2 : BOOL;
   TOP_CLAMP_FAULT_STN3 : BOOL;
   TOP_CLAMP_FAULT_STN4 : BOOL;
   TOP_CLAMP_OK_STN1 : BOOL;
   TOP_CLAMP_OK_STN2 : BOOL;
   TOP_CLAMP_OK_STN3 : BOOL;
   TOP_CLAMP_OK_STN4 : BOOL;
   TOP_CLAMP_ON_SEQ_STN1 : DINT;
   TOP_CLAMP_PR : REAL := 4.2654915;
   TOP_CLAMP_PR_CHK_STN1 : TIMER;
   TOP_CLAMP_PR_DEL : TIMER := (PRE := 6000);
   TOP_CLAMP_PR_SEL : BOOL := 1;
   TOP_CLAMP_PR_SEL_SET : BOOL;
   TOP_CLAMP_PR_SEL_SOL : ALIAS FOR REM:O.Data[1].6;
   TOP_CLAMP_PR_SEQ : CLAMP_FAULT := (CLAMP_PR_SEL := 1, CLAMP_PR := 4, CLAMP_2BAR_LL := 0.1, CLAMP_2BAR_HL := 3.5, CLAMP_4BAR_LL := 0.1, CLAMP_4BAR_HL := 4.5);
   TOP_CLAMP_PS_STN1 : ALIAS FOR Local:1:I.Data.12;
   TOP_CLAMP_PS_STN2 : ALIAS FOR Local:2:I.Data.1;
   TOP_CLAMP_PS_STN3 : ALIAS FOR Local:2:I.Data.6;
   TOP_CLAMP_PS_STN4 : ALIAS FOR Local:2:I.Data.11;
   TOP_CLAMP_SEL_STN1 : BOOL;
   TOP_CLAMP_SEL_STN2 : BOOL;
   TOP_CLAMP_SEL_STN3 : BOOL;
   TOP_CLAMP_SEL_STN4 : BOOL;
   TOP_CLAMP_SEQ_STN1 : DINT;
   TOP_CLAMP_SEQ_STN2 : DINT;
   TOP_CLAMP_SEQ_STN3 : DINT;
   TOP_CLAMP_SEQ_STN4 : DINT;
   TOP_CLAMP_SET_STN1 : BOOL;
   TOP_CLAMP_SET_STN2 : BOOL;
   TOP_CLAMP_SET_STN3 : BOOL;
   TOP_CLAMP_SET_STN4 : BOOL;
   TOP_CLAMP_SOL_STN1 : ALIAS FOR Local:1:O.Data.3;
   TOP_CLAMP_SOL_STN2 : ALIAS FOR Local:1:O.Data.11;
   TOP_CLAMP_SOL_STN3 : ALIAS FOR Local:3:O.Data.3;
   TOP_CLAMP_SOL_STN4 : ALIAS FOR Local:3:O.Data.11;
   TOP_CLAMP_X : REAL := 4.264;
   TOP_CLAMP_X1 : REAL;
   TOP_CLAMP_X2 : REAL := 5.718;
   TOP_CLAMP_Y1 : REAL;
   TOP_CLAMP_Y2 : REAL := 5.72;
   TOP_DECLAMP_AUTO_STN1 : BOOL;
   TOP_DECLAMP_AUTO_STN2 : BOOL;
   TOP_DECLAMP_AUTO_STN3 : BOOL;
   TOP_DECLAMP_AUTO_STN4 : BOOL;
   TOP_DECLAMP_BLK_STN1 : TOP_DECLAMP := (SET_SEQ_NO := 95, NEXT_SEQ_NO := 96, END_SEQ_NO := 96);
   TOP_DECLAMP_BLK_STN2 : TOP_DECLAMP := (SET_SEQ_NO := 95, NEXT_SEQ_NO := 96, END_SEQ_NO := 96);
   TOP_DECLAMP_BLK_STN3 : TOP_DECLAMP := (SET_SEQ_NO := 95, NEXT_SEQ_NO := 96, END_SEQ_NO := 96);
   TOP_DECLAMP_BLK_STN4 : TOP_DECLAMP := (SET_SEQ_NO := 95, NEXT_SEQ_NO := 96, END_SEQ_NO := 96);
   TOP_DECLAMP_OK_STN1 : BOOL;
   TOP_DECLAMP_OK_STN2 : BOOL;
   TOP_DECLAMP_OK_STN3 : BOOL;
   TOP_DECLAMP_OK_STN4 : BOOL;
   TOP_DECLAMP_RST_BLK_STN1 : TOP_DECLAMP := (SET_SEQ_NO := 114, NEXT_SEQ_NO := 115, END_SEQ_NO := 115);
   TOP_DECLAMP_rst_BLK_STN2 : TOP_DECLAMP := (SET_SEQ_NO := 114, NEXT_SEQ_NO := 115, END_SEQ_NO := 115);
   TOP_DECLAMP_RST_BLK_STN3 : TOP_DECLAMP := (SET_SEQ_NO := 114, NEXT_SEQ_NO := 115, END_SEQ_NO := 115);
   TOP_DECLAMP_RST_BLK_STN4 : TOP_DECLAMP := (SET_SEQ_NO := 114, NEXT_SEQ_NO := 115, END_SEQ_NO := 115);
   TOP_DECLAMP_SEQ_STN1 : DINT;
   TOP_DECLAMP_SEQ_STN2 : DINT;
   TOP_DECLAMP_SEQ_STN3 : DINT;
   TOP_DECLAMP_SEQ_STN4 : DINT;
   TOP_DECLAMP_SET_STN1 : BOOL;
   TOP_DECLAMP_SET_STN2 : BOOL;
   TOP_DECLAMP_SET_STN3 : BOOL;
   TOP_DECLAMP_SET_STN4 : BOOL;
   TOP_DECLAMP_SOL_STN1 : ALIAS FOR REM:O.Data[0].2;
   TOP_DECLAMP_SOL_STN2 : ALIAS FOR REM:O.Data[0].4;
   TOP_DECLAMP_SOL_STN3 : ALIAS FOR REM:O.Data[0].6;
   TOP_DECLAMP_SOL_STN4 : ALIAS FOR REM:O.Data[1].0;
   TOP_NOT_CLAMPED_STN1 : BOOL;
   TOP_NOT_DECLAMPED_STN1 : BOOL;
   TOP_NOT_DECLAMPED_STN2 : BOOL;
   TOP_NOT_DECLAMPED_STN3 : BOOL;
   TOP_NOT_DECLAMPED_STN4 : BOOL;
   TOP_PR : REAL;
   TOP_PR_SCL : SCP := (Y := 4.2654915, X := 4.264, X2 := 5.718, Y2 := 5.72);
   TOP_X1_MASTER : REAL;
   TOP_X2_MASTER : REAL;
   TOP_X_MASTER : REAL;
   TOP_Y1_MASTER : REAL;
   TOTAL_PASS_COUNT : DINT := 25;
   TRACE_FAULT_STN1 : BOOL;
   TRACE_ON_STN1 : BOOL := 1;
   TRACE_ON_STN2 : BOOL := 1;
   TRACE_ON_STN3 : BOOL := 1;
   TRACE_ON_STN4 : BOOL := 1;
   TS_STS_OP20A : DINT;
   TS_STS_OP20B : DINT;
   TS_STS_OP20C : DINT;
   TS_STS_OP20D : DINT := 3;
   TS_STS_STN1 : DINT;
   TS_STS_STN2 : DINT := 1;
   TS_STS_STN3 : DINT;
   TS_STS_STN4 : DINT;
   TS_TIMEOUT_FLT_STN1 : BOOL;
   TS_TIMEOUT_FLT_STN2 : BOOL;
   TS_TIMEOUT_FLT_STN3 : BOOL;
   TS_TIMEOUT_FLT_STN4 : BOOL;
   TS_TIMEOUT_STN1 : TS_TIMEOUT;
   TS_TIMEOUT_STN2 : TS_TIMEOUT;
   TS_TIMEOUT_STN3 : TS_TIMEOUT;
   TS_TIMEOUT_STN4 : TS_TIMEOUT;
   UNIT_SEL : DINT;
   UNLOCK_FAIL_BIN_PS_FLT : TIMER := (PRE := 3000);
   UNLOCK_FAIL_BIN_SOL : ALIAS FOR REM:O.Data[2].0;
   UNLOCK_FAULT_BIN_PS_FLT : TIMER := (PRE := 3000);
   UNLOCK_FAULT_BIN_SOL : ALIAS FOR REM:O.Data[2].1;
   USER_CHG : TIMER := (PRE := 1000);
   VIEW_PARAM : BOOL;
   VIEW_PARAM_OFF : TIMER := (PRE := 150);
   WHICH_STN_FAILED : DINT := 4;
   WHICH_STN_FAULTED : DINT := 4;
   WHICH_USER : INT;
   WORK_PR_CONS : REAL := 2677.0298;
   WORK_PR_PT : REAL := 2677.0298;
   WORK_PR_SCL : SCP := (Y := 2677.0298, X := 10.5, X1 := 1.999, X2 := 9.669, Y1 := 508.0, Y2 := 2465.0);
END_VAR

PROGRAM MainProgram   (* main routine MainRoutine *)
VAR
   ALIGN : SCP := (Y := 183439.48, X := 600.0, X2 := 785.0, Y2 := 240000.0);
   BOTTOM_NOT_CLAMPED_STN3 : BOOL;
   CLR_FLT_ONS_STN2 : BOOL;
   CLR_FLT_ONS_STN3 : BOOL;
   CLR_FLT_ONS_STN4 : BOOL;
   CONS_ONS1 : BOOL;
   CONS_ONS2 : BOOL;
   CONS_ONS3 : BOOL;
   CONS_ONS4 : BOOL;
   CONS_TEST_ON_DEL_STN3 : TIMER;
   CONS_TEST_ON_DEL_STN4 : TIMER;
   CYCLE_TIMER_STN2 : TIMER := (PRE := 99999);
   CYCLE_TIMER_STN3 : TIMER := (PRE := 99999);
   DFSDASFA : BOOL;
   DOOR_CLOSE_STS_STN1 : DINT;
   DOOR_CLOSE_STS_STN2 : DINT;
   DOOR_CLOSE_STS_STN3 : DINT;
   DOOR_CLOSE_STS_STN4 : DINT;
   DUMMY_VAL : REAL;
   EXHS_OK_DEL_STN1 : TIMER := (PRE := 500);
   EXHS_OK_DEL_STN2 : TIMER := (PRE := 500);
   EXHS_OK_DELSTN4 : TIMER := (PRE := 500);
   EXHS_VAL_HP_ON_STN2 : BOOL;
   EXHS_VAL_OFF_CE_STN1 : BOOL;
   EXHS_VAL_OFF_CE_STN2 : BOOL;
   EXHS_VAL_OFF_CE_STN3 : BOOL;
   EXHS_VAL_OFF_TE_STN1 : BOOL;
   EXHS_VAL_OFF_TE_STN2 : BOOL;
   EXHS_VAL_OFF_TE_STN3 : BOOL;
   FAIL_COMP_DROP_DEL : TIMER := (PRE := 1000);
   FAIL_COMP_DROPPED : BOOL;
   FAIL_FLUSHED : DINT := 4;
   FAULT_COMP_DROP_DEL : TIMER := (PRE := 1000);
   FAULT_COMP_DROPPED : BOOL;
   FAULT_COMP_SENSOR : ALIAS FOR Local:2:I.Data.30;
   FAULT_FIFO_DEL : TIMER := (PRE := 250, ACC := 251);
   FAULT_FLUSHED : DINT := 4;
   fdsdf : COUNTER := (PRE := 9999, ACC := 6387);
   FIFO_INDEX : DINT;
   FLT_CLEAR_ONS_STN4 : BOOL;
   FLUSH_BIN_DROP : TIMER := (PRE := 100, ACC := 103, EN := 1, DN := 1);
   FLUSH_FAIL_BIN_DROP : TIMER := (PRE := 100, ACC := 103, EN := 1, DN := 1);
   GET_FIRST_FAULTED : DINT;
        .0   // STN1 FAULTED
        .2   // STN3 FAULTED
        .3   // STN4 FAULTED
        .1   // STN2 FAULTED
   GOTO_FAIL_BIN_STN1 : DINT;
   GOTO_FAULT_BIN_STN3 : DINT;
   GOTO_FAULT_BIN_STN4 : DINT;
   INDV_LTEST_ON_STN1 : BOOL;
   INDV_LTEST_ON_STN2 : BOOL;
   INDV_LTEST_ON_STN3 : BOOL;
   INDV_LTEST_ON_STN4 : BOOL;
   LOCK_FAULT_BIN : BOOL;
   ONS1 : BOOL;
   ONS10 : BOOL;
   ONS104 : BOOL := 1;
   ONS11 : BOOL;
   ONS12 : BOOL;
   ONS13 : BOOL;
   ONS14 : BOOL;
   ONS15 : BOOL;
   ONS16 : BOOL;
   ONS17 : BOOL;
   ONS18 : BOOL;
   ONS19 : BOOL;
   ONS2 : BOOL;
   ONS20 : BOOL;
   ONS21 : BOOL;
   ONS22 : BOOL;
   ONS23 : BOOL;
   ONS24 : BOOL;
   ONS25 : BOOL;
   ONS26 : BOOL;
   ONS27 : BOOL;
   ONS28 : BOOL;
   ONS29 : BOOL;
   ONS3 : BOOL;
   ONS30 : BOOL;
   ONS31 : BOOL;
   ONS32 : BOOL;
   ONS33 : BOOL;
   ONS35 : BOOL;
   ONS36 : BOOL;
   ONS37 : BOOL;
   ONS38 : BOOL;
   ONS39 : BOOL;
   ONS4 : BOOL;
   ONS40 : BOOL;
   ONS41 : BOOL := 1;
   ONS42 : BOOL;
   ONS43 : BOOL := 1;
   ONS44 : BOOL := 1;
   ONS45 : BOOL := 1;
   ONS46 : BOOL := 1;
   ONS47 : BOOL;
   ONS48 : BOOL;
   ONS49 : BOOL;
   ONS50 : BOOL;
   ONS51 : BOOL;
   ONS52 : BOOL;
   ONS53 : BOOL := 1;
   ONS54 : BOOL;
   ONS55 : BOOL;
   ONS56 : BOOL;
   ONS57 : BOOL;
   ONS58 : BOOL;
   ONS59 : BOOL;
   ONS6 : BOOL;
   ONS60 : BOOL;
   ONS61 : BOOL;
   ONS62 : BOOL;
   ONS63 : BOOL := 1;
   ONS64 : BOOL;
   ONS65 : BOOL;
   ONS66 : BOOL := 1;
   ONS67 : BOOL;
   ONS68 : BOOL;
   ONS69 : BOOL;
   ONS7 : BOOL;
   ONS70 : BOOL;
   ONS71 : BOOL := 1;
   ONS72 : BOOL := 1;
   ONS73 : BOOL := 1;
   ONS74 : BOOL := 1;
   ONS75 : BOOL := 1;
   ONS8 : BOOL;
   ONS9 : BOOL := 1;
   ONS_100 : BOOL;
   ONS_101 : BOOL;
   ONS_102 : BOOL;
   ONS_103 : BOOL := 1;
   ONS_70 : BOOL := 1;
   ONS_71 : BOOL := 1;
   ONS_72 : BOOL := 1;
   ONS_74 : BOOL;
   ONS_75 : BOOL;
   ONS_76 : BOOL;
   ONS_77 : BOOL;
   ONS_78 : BOOL;
   ONS_79 : BOOL;
   ONS_80 : BOOL;
   ONS_81 : BOOL;
   ONS_82 : BOOL;
   ONS_83 : BOOL;
   ONS_84 : BOOL;
   ONS_85 : BOOL;
   ONS_86 : BOOL;
   ONS_87 : BOOL;
   ONS_88 : BOOL;
   ONS_89 : BOOL;
   ONS_90 : BOOL;
   ONS_91 : BOOL;
   ONS_92 : BOOL;
   ONS_93 : BOOL;
   ONS_94 : BOOL := 1;
   ONS_95 : BOOL;
   ONS_96 : BOOL;
   ONS_97 : BOOL;
   ONS_98 : BOOL;
   ONS_99 : BOOL;
   PASS_COUNTER_STN1 : COUNTER := (PRE := 9999, ACC := 4);
   PASS_COUNTER_STN2 : COUNTER := (PRE := 9999, ACC := 9);
   PASS_COUNTER_STN3 : COUNTER := (PRE := 9999, ACC := 12);
   PASS_COUNTER_STN4 : COUNTER := (PRE := 9999);
   RST_DOOR_NOT_OPENED_STN3 : BOOL;
   RST_DOOR_OPEN_OK_STN1 : BOOL;
   RST_DOOR_OPEN_OK_STN2 : BOOL;
   RST_DOOR_OPEN_OK_STN3 : BOOL;
   RST_FLT_CLR_ONS_STN2 : BOOL;
   RST_FLT_CLR_ONS_STN3 : BOOL;
   RST_TOP_NOT_DECLAMPED_STN1 : BOOL;
   RST_TOP_NOT_DECLAMPED_STN2 : BOOL;
   RST_TOP_NOT_DECLAMPED_STN3 : BOOL;
   RST_TOP_NOT_DECLAMPED_STN4 : BOOL;
   TEST_INIT_DEL_STN2 : TIMER := (PRE := 250);
   TEST_INIT_DEL_STN3 : TIMER := (PRE := 250);
   TEST_INIT_DEL_STN4 : TIMER := (PRE := 250);
   TEST_VAL_OFF_HP_STN1 : BOOL;
   TIME1 : TIMER := (PRE := 183439, ACC := 61146, EN := 1, DN := 1);
   TOP_NOT_CLAMPED_STN2 : BOOL;
   TOP_NOT_CLAMPED_STN3 : BOOL;
   TOP_NOT_CLAMPED_STN4 : BOOL;
END_VAR
